  Call Extruder(6734.21438)
  MoveL 616 to (16.69, 20.93, 35) mm, rotated rx -180 ry 0 rz 180 deg; joints [-158.019, -62.995, -84.833, 25.494, 60.412, -13.249]
  Call Extruder(6743.57930)
  MoveL 617 to (11.61, 24.11, 35) mm, rotated rx -180 ry 0 rz 180 deg; joints [-157.299, -62.811, -85.449, 26.193, 60.967, -13.427]
  Call Extruder(6752.94410)
  MoveL 618 to (5.96, 26.09, 35) mm, rotated rx 180 ry 0 rz 180 deg; joints [-156.697, -62.583, -86.227, 26.726, 61.599, -13.468]
  Call Extruder(6762.30921)
  MoveL 619 to (0, 26.77, 35) mm, rotated rx -180 ry 0 rz 180 deg; joints [-156.245, -62.323, -87.131, 27.069, 62.279, -13.372]
  Call Extruder(6771.67431)
  MoveL 620 to (-5.96, 26.09, 35) mm, rotated rx 180 ry 0 rz 180 deg; joints [-155.969, -62.047, -88.117, 27.203, 62.974, -13.147]
  Call Extruder(6781.03910)
  MoveL 621 to (-11.61, 24.12, 35) mm, rotated rx 180 ry 0 rz 180 deg; joints [-155.891, -61.768, -89.137, 27.118, 63.651, -12.806]
  Call Extruder(6790.40402)
  MoveL 622 to (-16.69, 20.93, 35) mm, rotated rx 180 ry 0 rz -180 deg; joints [-156.025, -61.503, -90.14, 26.81, 64.279, -12.37]
  Call Extruder(6799.76923)
  MoveL 623 to (-20.93, 16.69, 35) mm, rotated rx 180 ry 0 rz 180 deg; joints [-156.374, -61.262, -91.076, 26.284, 64.828, -11.863]
  Call Extruder(6809.13414)
  MoveL 624 to (-24.11, 11.61, 35) mm, rotated rx -180 ry 0 rz 180 deg; joints [-156.928, -61.058, -91.897, 25.56, 65.271, -11.314]
  Call Extruder(6818.49894)
  MoveL 625 to (-26.09, 5.96, 35) mm, rotated rx -180 ry 0 rz 180 deg; joints [-157.665, -60.897, -92.558, 24.667, 65.583, -10.749]
  Call Extruder(6827.86405)
  MoveL 626 to (-26.77, 0, 35) mm, rotated rx 180 ry 0 rz 180 deg; joints [-158.546, -60.787, -93.024, 23.65, 65.748, -10.198]
  Call Extruder(6832.65278)
  MoveL 627 to (-26.42, -3.05, 35) mm, rotated rx -180 ry 0 rz 180 deg; joints [-159.044, -60.757, -93.152, 23.095, 65.75, -9.934]
  Set speed (130.0 mm/s)
  MoveL 628 to (-41.86, -6.29, 35) mm, rotated rx 180 ry 0 rz -180 deg; joints [-158.606, -60.2, -95.665, 23.234, 67.622, -9.283]
  Call Extruder(6837.65063)
  Set speed (60.0 mm/s)
  MoveL 629 to (-41.5, -9.47, 35) mm, rotated rx 180 ry 0 rz 180 deg; joints [-159.151, -60.173, -95.794, 22.635, 67.63, -9.018]
  Call Extruder(6852.54627)
  MoveL 630 to (-38.36, -18.47, 35) mm, rotated rx 180 ry 0 rz -180 deg; joints [-160.835, -60.169, -95.813, 20.831, 67.39, -8.322]
  Call Extruder(6867.44213)
  MoveL 631 to (-33.29, -26.54, 35) mm, rotated rx 180 ry 0 rz -180 deg; joints [-162.466, -60.245, -95.451, 19.121, 66.892, -7.748]
  Call Extruder(6882.33794)
  MoveL 632 to (-26.54, -33.28, 35) mm, rotated rx -180 ry 0 rz -180 deg; joints [-163.93, -60.4, -94.729, 17.616, 66.162, -7.313]
  Call Extruder(6897.23380)
  MoveL 633 to (-18.47, -38.36, 35) mm, rotated rx 180 ry 0 rz 180 deg; joints [-165.137, -60.632, -93.69, 16.408, 65.24, -7.031]
  Call Extruder(6912.12945)
  MoveL 634 to (-9.47, -41.5, 35) mm, rotated rx 180 ry 0 rz 180 deg; joints [-166.024, -60.937, -92.392, 15.563, 64.178, -6.917]
  Call Extruder(6927.02533)
  MoveL 635 to (0, -42.57, 35) mm, rotated rx 180 ry 0 rz 180 deg; joints [-166.562, -61.305, -90.908, 15.114, 63.036, -6.982]
  Call Extruder(6928.24069)
  MoveL 636 to (0.77, -42.49, 35) mm, rotated rx 180 ry 0 rz 180 deg; joints [-166.577, -61.338, -90.779, 15.11, 62.942, -7.002]
  Call Extruder(6941.92120)
  MoveL 637 to (9.47, -41.51, 35) mm, rotated rx 180 ry 0 rz 180 deg; joints [-166.745, -61.721, -89.315, 15.069, 61.877, -7.233]
  Call Extruder(6956.81686)
  MoveL 638 to (18.47, -38.36, 35) mm, rotated rx 180 ry 0 rz 180 deg; joints [-166.591, -62.165, -87.694, 15.412, 60.761, -7.669]
  Call Extruder(6971.71270)
  MoveL 639 to (26.54, -33.28, 35) mm, rotated rx 180 ry 0 rz 180 deg; joints [-166.133, -62.613, -86.123, 16.109, 59.745, -8.279]
  Call Extruder(6986.60852)
  MoveL 640 to (33.29, -26.54, 35) mm, rotated rx -180 ry 0 rz 180 deg; joints [-165.409, -63.041, -84.679, 17.113, 58.88, -9.041]
  Call Extruder(7001.50437)
  MoveL 641 to (38.36, -18.47, 35) mm, rotated rx 180 ry 0 rz 180 deg; joints [-164.468, -63.423, -83.43, 18.364, 58.208, -9.92]
  Call Extruder(7016.40003)
  MoveL 642 to (41.5, -9.47, 35) mm, rotated rx 180 ry 0 rz 180 deg; joints [-163.355, -63.734, -82.433, 19.795, 57.761, -10.868]
  Call Extruder(7031.29590)
  MoveL 643 to (42.57, 0, 35) mm, rotated rx 180 ry 0 rz 180 deg; joints [-162.12, -63.955, -81.735, 21.334, 57.558, -11.833]
  Call Extruder(7046.19177)
  MoveL 644 to (41.5, 9.47, 35) mm, rotated rx 180 ry 0 rz 180 deg; joints [-160.81, -64.073, -81.369, 22.909, 57.606, -12.757]
  Call Extruder(7061.08744)
  MoveL 645 to (38.36, 18.47, 35) mm, rotated rx 180 ry 0 rz 180 deg; joints [-159.475, -64.078, -81.351, 24.45, 57.9, -13.583]
  Call Extruder(7075.98328)
  MoveL 646 to (33.29, 26.54, 35) mm, rotated rx 180 ry 0 rz 180 deg; joints [-158.16, -63.972, -81.683, 25.892, 58.42, -14.262]
  Call Extruder(7090.87910)
  MoveL 647 to (26.54, 33.28, 35) mm, rotated rx -180 ry 0 rz 180 deg; joints [-156.916, -63.76, -82.349, 27.178, 59.139, -14.755]
  Call Extruder(7105.77495)
  MoveL 648 to (18.47, 38.36, 35) mm, rotated rx -180 ry 0 rz -180 deg; joints [-155.789, -63.457, -83.319, 28.259, 60.018, -15.035]
  Call Extruder(7120.67061)
  MoveL 649 to (9.47, 41.51, 35) mm, rotated rx -180 ry 0 rz 180 deg; joints [-154.828, -63.081, -84.546, 29.094, 61.015, -15.091]
  Call Extruder(7135.56648)
  MoveL 650 to (0, 42.57, 35) mm, rotated rx 180 ry 0 rz 180 deg; joints [-154.081, -62.657, -85.973, 29.648, 62.083, -14.922]
  Call Extruder(7150.46236)
  MoveL 651 to (-9.47, 41.51, 35) mm, rotated rx 180 ry 0 rz 180 deg; joints [-153.594, -62.209, -87.534, 29.892, 63.173, -14.543]
  Call Extruder(7165.35801)
  MoveL 652 to (-18.47, 38.36, 35) mm, rotated rx 180 ry 0 rz 180 deg; joints [-153.408, -61.764, -89.154, 29.804, 64.237, -13.98]
  Call Extruder(7180.25386)
  MoveL 653 to (-26.54, 33.28, 35) mm, rotated rx 180 ry 0 rz -180 deg; joints [-153.557, -61.344, -90.754, 29.369, 65.228, -13.268]
  Call Extruder(7195.14968)
  MoveL 654 to (-33.29, 26.54, 35) mm, rotated rx -180 ry 0 rz 180 deg; joints [-154.059, -60.971, -92.252, 28.585, 66.101, -12.448]
  Call Extruder(7210.04552)
  MoveL 655 to (-38.36, 18.47, 35) mm, rotated rx 180 ry 0 rz 180 deg; joints [-154.913, -60.659, -93.571, 27.468, 66.813, -11.568]
  Call Extruder(7224.94118)
  MoveL 656 to (-41.5, 9.47, 35) mm, rotated rx 180 ry 0 rz 180 deg; joints [-156.091, -60.419, -94.639, 26.056, 67.325, -10.674]
  Call Extruder(7239.83706)
  MoveL 657 to (-42.57, 0, 35) mm, rotated rx -180 ry 0 rz -180 deg; joints [-157.533, -60.257, -95.395, 24.414, 67.605, -9.812]
  Call Extruder(7247.39133)
  MoveL 658 to (-42.03, -4.8, 35) mm, rotated rx 180 ry 0 rz 180 deg; joints [-158.35, -60.213, -95.603, 23.515, 67.618, -9.407]
  Set speed (130.0 mm/s)
  MoveL 659 to (-54.1, -7.67, 35) mm, rotated rx -180 ry 0 rz -180 deg; joints [-158.024, -59.828, -97.542, 23.615, 69.095, -8.867]
  Call Extruder(7251.46397)
  Set speed (30.0 mm/s)
  MoveL 660 to (-53.59, -12.23, 35) mm, rotated rx 180 ry 0 rz -180 deg; joints [-158.835, -59.793, -97.729, 22.734, 69.112, -8.497]
  Call Extruder(7262.39410)
  MoveL 661 to (-49.52, -23.85, 35) mm, rotated rx 180 ry 0 rz 180 deg; joints [-161.095, -59.788, -97.754, 20.333, 68.814, -7.628]
  Call Extruder(7273.32438)
  MoveL 662 to (-42.98, -34.27, 35) mm, rotated rx 180 ry 0 rz 180 deg; joints [-163.275, -59.878, -97.277, 18.059, 68.172, -6.913]
  Call Extruder(7284.25450)
  MoveL 663 to (-34.27, -42.98, 35) mm, rotated rx -180 ry 0 rz 180 deg; joints [-165.21, -60.064, -96.329, 16.073, 67.22, -6.366]
  Call Extruder(7295.18479)
  MoveL 664 to (-23.85, -49.53, 35) mm, rotated rx 180 ry 0 rz -180 deg; joints [-166.774, -60.347, -94.97, 14.502, 66.014, -6.003]
  Call Extruder(7306.11492)
  MoveL 665 to (-12.23, -53.59, 35) mm, rotated rx 180 ry 0 rz 180 deg; joints [-167.889, -60.727, -93.28, 13.427, 64.627, -5.841]
  Call Extruder(7317.04514)
  MoveL 666 to (0, -54.97, 35) mm, rotated rx 180 ry 0 rz 180 deg; joints [-168.526, -61.192, -91.354, 12.884, 63.139, -5.9]
  Call Extruder(7318.96829)
  MoveL 667 to (2.15, -54.73, 35) mm, rotated rx 180 ry 0 rz -180 deg; joints [-168.557, -61.283, -90.994, 12.88, 62.874, -5.952]
  Call Extruder(7327.97536)
  MoveL 668 to (12.23, -53.59, 35) mm, rotated rx -180 ry 0 rz 180 deg; joints [-168.697, -61.726, -89.294, 12.87, 61.634, -6.196]
  Call Extruder(7338.90550)
  MoveL 669 to (23.85, -49.53, 35) mm, rotated rx 180 ry 0 rz 180 deg; joints [-168.436, -62.303, -87.203, 13.358, 60.189, -6.732]
  Call Extruder(7349.83578)
  MoveL 670 to (34.27, -42.98, 35) mm, rotated rx 180 ry 0 rz -180 deg; joints [-167.797, -62.89, -85.184, 14.295, 58.877, -7.503]
  Call Extruder(7360.76590)
  MoveL 671 to (42.98, -34.27, 35) mm, rotated rx 180 ry 0 rz 180 deg; joints [-166.837, -63.454, -83.329, 15.618, 57.763, -8.481]
  Call Extruder(7371.69618)
  MoveL 672 to (49.53, -23.85, 35) mm, rotated rx -180 ry 0 rz 180 deg; joints [-165.618, -63.958, -81.725, 17.247, 56.9, -9.622]
  Call Extruder(7382.62632)
  MoveL 673 to (53.59, -12.23, 35) mm, rotated rx 180 ry 0 rz -180 deg; joints [-164.2, -64.372, -80.446, 19.097, 56.33, -10.865]
  Call Extruder(7393.55654)
  MoveL 674 to (54.97, 0, 35) mm, rotated rx -180 ry 0 rz 180 deg; joints [-162.641, -64.667, -79.551, 21.074, 56.077, -12.137]
  Call Extruder(7404.48676)
  MoveL 675 to (53.59, 12.23, 35) mm, rotated rx -180 ry 0 rz 180 deg; joints [-160.996, -64.823, -79.081, 23.085, 56.149, -13.356]
  Call Extruder(7415.41691)
  MoveL 676 to (49.52, 23.85, 35) mm, rotated rx 180 ry 0 rz -180 deg; joints [-159.322, -64.831, -79.058, 25.041, 56.538, -14.445]
  Call Extruder(7426.34718)
  MoveL 677 to (42.98, 34.27, 35) mm, rotated rx -180 ry 0 rz 180 deg; joints [-157.673, -64.689, -79.485, 26.863, 57.217, -15.337]
  Call Extruder(7437.27731)
  MoveL 678 to (34.27, 42.98, 35) mm, rotated rx 180 ry 0 rz 180 deg; joints [-156.102, -64.407, -80.339, 28.484, 58.149, -15.979]
  Call Extruder(7448.20758)
  MoveL 679 to (23.85, 49.52, 35) mm, rotated rx -180 ry 0 rz 180 deg; joints [-154.667, -64.004, -81.583, 29.848, 59.282, -16.337]
  Call Extruder(7459.13773)
  MoveL 680 to (12.23, 53.59, 35) mm, rotated rx -180 ry 0 rz 180 deg; joints [-153.426, -63.507, -83.157, 30.909, 60.562, -16.397]
  Call Extruder(7470.06795)
  MoveL 681 to (0, 54.97, 35) mm, rotated rx 180 ry 0 rz 180 deg; joints [-152.438, -62.948, -84.991, 31.628, 61.928, -16.163]
  Call Extruder(7480.99817)
  MoveL 682 to (-12.23, 53.59, 35) mm, rotated rx -180 ry 0 rz 180 deg; joints [-151.764, -62.361, -86.998, 31.97, 63.32, -15.655]
  Call Extruder(7491.92830)
  MoveL 683 to (-23.85, 49.52, 35) mm, rotated rx 180 ry 0 rz 180 deg; joints [-151.463, -61.782, -89.086, 31.904, 64.68, -14.909]
  Call Extruder(7502.85859)
  MoveL 684 to (-34.27, 42.98, 35) mm, rotated rx -180 ry 0 rz 180 deg; joints [-151.589, -61.243, -91.154, 31.401, 65.949, -13.97]
  Call Extruder(7513.78871)
  MoveL 685 to (-42.98, 34.27, 35) mm, rotated rx 180 ry 0 rz -180 deg; joints [-152.179, -60.769, -93.098, 30.446, 67.074, -12.897]
  Call Extruder(7524.71899)
  MoveL 686 to (-49.52, 23.85, 35) mm, rotated rx 180 ry 0 rz 180 deg; joints [-153.248, -60.381, -94.816, 29.044, 68, -11.751]
  Call Extruder(7535.64913)
  MoveL 687 to (-53.59, 12.23, 35) mm, rotated rx 180 ry 0 rz 180 deg; joints [-154.769, -60.087, -96.212, 27.231, 68.678, -10.599]
  Call Extruder(7546.57935)
  MoveL 688 to (-54.97, 0, 35) mm, rotated rx -180 ry 0 rz -180 deg; joints [-156.673, -59.892, -97.203, 25.087, 69.06, -9.498]
  Call Extruder(7552.10496)
  MoveL 689 to (-54.27, -6.18, 35) mm, rotated rx -180 ry 0 rz 180 deg; joints [-157.76, -59.84, -97.478, 23.902, 69.088, -8.989]
  Set speed (130.0 mm/s)
  MoveL 690 to (-49.9, -9.51, 35) mm, rotated rx -180 ry 0 rz -180 deg; joints [-158.616, -59.924, -97.035, 23.05, 68.627, -8.815]
  MoveL 691 to (2.97, -12.99, 35) mm, rotated rx 180 ry 0 rz -180 deg; joints [-162.152, -61.783, -89.081, 20.235, 62.39, -9.695]
  Call Extruder(7556.76854)
  Set speed (80.0 mm/s)
  MoveL 692 to (5.78, -12.01, 35) mm, rotated rx -180 ry 0 rz 180 deg; joints [-162.141, -61.921, -88.573, 20.316, 62.045, -9.846]
  Call Extruder(7561.43216)
  MoveL 693 to (8.31, -10.42, 35) mm, rotated rx -180 ry 0 rz -180 deg; joints [-162.027, -62.058, -88.077, 20.51, 61.728, -10.048]
  Call Extruder(7566.09635)
  MoveL 694 to (10.42, -8.31, 35) mm, rotated rx 180 ry 0 rz 180 deg; joints [-161.819, -62.185, -87.619, 20.805, 61.455, -10.291]
  Call Extruder(7570.75998)
  MoveL 695 to (12.01, -5.78, 35) mm, rotated rx 180 ry 0 rz 180 deg; joints [-161.529, -62.298, -87.221, 21.187, 61.241, -10.564]
  Call Extruder(7575.42355)
  MoveL 696 to (12.99, -2.97, 35) mm, rotated rx 180 ry 0 rz -180 deg; joints [-161.171, -62.388, -86.903, 21.634, 61.096, -10.852]
  Call Extruder(7580.08750)
  MoveL 697 to (13.33, 0, 35) mm, rotated rx 180 ry 0 rz 180 deg; joints [-160.763, -62.452, -86.68, 22.124, 61.026, -11.141]
  Call Extruder(7584.75146)
  MoveL 698 to (13, 2.97, 35) mm, rotated rx 180 ry 0 rz 180 deg; joints [-160.324, -62.486, -86.563, 22.634, 61.035, -11.416]
  Call Extruder(7589.41503)
  MoveL 699 to (12.01, 5.78, 35) mm, rotated rx 180 ry 0 rz -180 deg; joints [-159.874, -62.488, -86.557, 23.139, 61.121, -11.661]
  Call Extruder(7594.07865)
  MoveL 700 to (10.42, 8.31, 35) mm, rotated rx -180 ry 0 rz 180 deg; joints [-159.432, -62.457, -86.663, 23.615, 61.28, -11.864]
  Call Extruder(7598.74284)
  MoveL 701 to (8.31, 10.42, 35) mm, rotated rx 180 ry 0 rz 180 deg; joints [-159.021, -62.396, -86.876, 24.041, 61.505, -12.014]
  Call Extruder(7603.40647)
  MoveL 702 to (5.78, 12.01, 35) mm, rotated rx 180 ry 0 rz 180 deg; joints [-158.657, -62.308, -87.186, 24.396, 61.782, -12.103]
  Call Extruder(7608.07004)
  MoveL 703 to (2.97, 12.99, 35) mm, rotated rx -180 ry 0 rz 180 deg; joints [-158.359, -62.197, -87.577, 24.663, 62.1, -12.126]
  Call Extruder(7612.73400)
  MoveL 704 to (0, 13.33, 35) mm, rotated rx 180 ry 0 rz -180 deg; joints [-158.143, -62.071, -88.03, 24.831, 62.442, -12.083]
  Call Extruder(7617.39795)
  MoveL 705 to (-2.97, 12.99, 35) mm, rotated rx -180 ry 0 rz 180 deg; joints [-158.019, -61.935, -88.523, 24.889, 62.792, -11.977]
  Call Extruder(7622.06151)
  MoveL 706 to (-5.78, 12.01, 35) mm, rotated rx 180 ry 0 rz 180 deg; joints [-157.997, -61.797, -89.031, 24.834, 63.132, -11.813]
  Call Extruder(7626.72515)
  MoveL 707 to (-8.31, 10.42, 35) mm, rotated rx -180 ry 0 rz 180 deg; joints [-158.08, -61.663, -89.53, 24.666, 63.447, -11.601]
  Call Extruder(7631.38934)
  MoveL 708 to (-10.42, 8.31, 35) mm, rotated rx 180 ry 0 rz 180 deg; joints [-158.266, -61.541, -89.993, 24.392, 63.72, -11.352]
  Call Extruder(7636.05296)
  MoveL 709 to (-12.01, 5.78, 35) mm, rotated rx 180 ry 0 rz 180 deg; joints [-158.549, -61.436, -90.398, 24.023, 63.938, -11.079]
  Call Extruder(7640.71653)
  MoveL 710 to (-13, 2.97, 35) mm, rotated rx -180 ry 0 rz -180 deg; joints [-158.913, -61.352, -90.723, 23.577, 64.09, -10.796]
  Call Extruder(7645.38049)
  MoveL 711 to (-13.33, 0, 35) mm, rotated rx -180 ry 0 rz 180 deg; joints [-159.341, -61.294, -90.952, 23.077, 64.168, -10.517]
  Call Extruder(7650.04444)
  MoveL 712 to (-13, -2.97, 35) mm, rotated rx -180 ry 0 rz 180 deg; joints [-159.811, -61.263, -91.072, 22.547, 64.166, -10.255]
  Call Extruder(7654.70800)
  MoveL 713 to (-12.01, -5.78, 35) mm, rotated rx -180 ry 0 rz 180 deg; joints [-160.294, -61.262, -91.078, 22.017, 64.085, -10.022]
  Call Extruder(7659.37164)
  MoveL 714 to (-10.42, -8.31, 35) mm, rotated rx 180 ry 0 rz 180 deg; joints [-160.766, -61.289, -90.969, 21.515, 63.928, -9.829]
  Call Extruder(7664.03583)
  MoveL 715 to (-8.31, -10.42, 35) mm, rotated rx 180 ry 0 rz 180 deg; joints [-161.2, -61.345, -90.75, 21.068, 63.702, -9.685]
  Call Extruder(7668.69946)
  MoveL 716 to (-5.78, -12.01, 35) mm, rotated rx 180 ry 0 rz 180 deg; joints [-161.572, -61.426, -90.434, 20.7, 63.421, -9.597]
  Call Extruder(7673.36302)
  MoveL 717 to (-2.97, -13, 35) mm, rotated rx 180 ry 0 rz 180 deg; joints [-161.863, -61.53, -90.036, 20.431, 63.097, -9.568]
  Call Extruder(7678.02699)
  MoveL 718 to (0, -13.33, 35) mm, rotated rx -180 ry 0 rz -180 deg; joints [-162.059, -61.651, -89.577, 20.274, 62.747, -9.601]
  Call Extruder(7682.69093)
  MoveL 719 to (2.97, -12.99, 35) mm, rotated rx 180 ry 0 rz -180 deg; joints [-162.152, -61.783, -89.081, 20.235, 62.39, -9.695]
  Set speed (130.0 mm/s)
  MoveL 720 to (2.97, -12.99, 40) mm, rotated rx 180 ry 0 rz -180 deg; joints [-162.152, -61.016, -89.511, 20.297, 62.074, -9.827]
  MoveL 721 to (-26.25, -4.54, 40) mm, rotated rx 180 ry 0 rz -180 deg; joints [-159.288, -59.949, -93.651, 22.886, 65.424, -9.957]
  Call Extruder(7684.92356)
  Set speed (60.0 mm/s)
  MoveL 722 to (-26.09, -5.96, 40) mm, rotated rx 180 ry 0 rz 180 deg; joints [-159.522, -59.936, -93.708, 22.625, 65.424, -9.834]
  Call Extruder(7694.28835)
  MoveL 723 to (-24.11, -11.61, 40) mm, rotated rx 180 ry 0 rz 180 deg; joints [-160.532, -59.933, -93.72, 21.528, 65.264, -9.373]
  Call Extruder(7703.65327)
  MoveL 724 to (-20.93, -16.69, 40) mm, rotated rx 180 ry 0 rz -180 deg; joints [-161.513, -59.986, -93.496, 20.488, 64.949, -8.991]
  Call Extruder(7713.01847)
  MoveL 725 to (-16.69, -20.93, 40) mm, rotated rx 180 ry 0 rz 180 deg; joints [-162.406, -60.095, -93.05, 19.567, 64.494, -8.702]
  Call Extruder(7722.38339)
  MoveL 726 to (-11.61, -24.12, 40) mm, rotated rx 180 ry 0 rz 180 deg; joints [-163.159, -60.254, -92.405, 18.817, 63.923, -8.519]
  Call Extruder(7731.74818)
  MoveL 727 to (-5.96, -26.09, 40) mm, rotated rx 180 ry 0 rz 180 deg; joints [-163.733, -60.46, -91.597, 18.278, 63.267, -8.451]
  Call Extruder(7741.11329)
  MoveL 728 to (0, -26.77, 40) mm, rotated rx 180 ry 0 rz 180 deg; joints [-164.103, -60.703, -90.669, 17.977, 62.561, -8.504]
  Call Extruder(7745.37891)
  MoveL 729 to (2.71, -26.46, 40) mm, rotated rx -180 ry 0 rz -180 deg; joints [-164.174, -60.824, -90.215, 17.951, 62.234, -8.583]
  Call Extruder(7750.47839)
  MoveL 730 to (5.96, -26.09, 40) mm, rotated rx 180 ry 0 rz -180 deg; joints [-164.258, -60.973, -89.668, 17.922, 61.843, -8.677]
  Call Extruder(7759.84319)
  MoveL 731 to (11.61, -24.11, 40) mm, rotated rx 180 ry 0 rz 180 deg; joints [-164.201, -61.256, -88.646, 18.111, 61.149, -8.968]
  Call Extruder(7769.20811)
  MoveL 732 to (16.69, -20.93, 40) mm, rotated rx 180 ry 0 rz 180 deg; joints [-163.944, -61.539, -87.653, 18.526, 60.516, -9.365]
  Call Extruder(7778.57331)
  MoveL 733 to (20.93, -16.69, 40) mm, rotated rx -180 ry 0 rz 180 deg; joints [-163.508, -61.806, -86.738, 19.14, 59.975, -9.852]
  Call Extruder(7787.93823)
  MoveL 734 to (24.12, -11.61, 40) mm, rotated rx -180 ry 0 rz 180 deg; joints [-162.92, -62.042, -85.944, 19.919, 59.553, -10.405]
  Call Extruder(7797.30303)
  MoveL 735 to (26.09, -5.96, 40) mm, rotated rx -180 ry 0 rz -180 deg; joints [-162.209, -62.234, -85.311, 20.821, 59.271, -10.996]
  Call Extruder(7806.66813)
  MoveL 736 to (26.77, 0, 40) mm, rotated rx -180 ry 0 rz -180 deg; joints [-161.41, -62.37, -84.867, 21.8, 59.14, -11.594]
  Call Extruder(7816.03323)
  MoveL 737 to (26.09, 5.96, 40) mm, rotated rx -180 ry 0 rz 180 deg; joints [-160.556, -62.441, -84.634, 22.81, 59.167, -12.164]
  Call Extruder(7825.39804)
  MoveL 738 to (24.12, 11.61, 40) mm, rotated rx 180 ry 0 rz 180 deg; joints [-159.683, -62.445, -84.623, 23.804, 59.348, -12.675]
  Call Extruder(7834.76295)
  MoveL 739 to (20.93, 16.69, 40) mm, rotated rx -180 ry 0 rz 180 deg; joints [-158.826, -62.38, -84.834, 24.738, 59.672, -13.097]
  Call Extruder(7844.12816)
  MoveL 740 to (16.69, 20.93, 40) mm, rotated rx -180 ry 0 rz 180 deg; joints [-158.019, -62.25, -85.258, 25.573, 60.123, -13.408]
  Call Extruder(7853.49307)
  MoveL 741 to (11.61, 24.11, 40) mm, rotated rx -180 ry 0 rz 180 deg; joints [-157.299, -62.063, -85.874, 26.272, 60.678, -13.59]
  Call Extruder(7862.85787)
  MoveL 742 to (5.96, 26.09, 40) mm, rotated rx 180 ry 0 rz 180 deg; joints [-156.697, -61.831, -86.653, 26.805, 61.308, -13.635]
  Call Extruder(7872.22298)
  MoveL 743 to (0, 26.77, 40) mm, rotated rx -180 ry 0 rz 180 deg; joints [-156.245, -61.566, -87.558, 27.148, 61.985, -13.542]
  Call Extruder(7881.58808)
  MoveL 744 to (-5.96, 26.09, 40) mm, rotated rx 180 ry 0 rz 180 deg; joints [-155.969, -61.284, -88.546, 27.282, 62.677, -13.318]
  Call Extruder(7890.95287)
  MoveL 745 to (-11.61, 24.12, 40) mm, rotated rx -180 ry 0 rz 180 deg; joints [-155.891, -61, -89.567, 27.195, 63.35, -12.978]
  Call Extruder(7900.31779)
  MoveL 746 to (-16.69, 20.93, 40) mm, rotated rx 180 ry 0 rz -180 deg; joints [-156.025, -60.729, -90.572, 26.885, 63.974, -12.542]
  Call Extruder(7909.68300)
  MoveL 747 to (-20.93, 16.69, 40) mm, rotated rx 180 ry 0 rz -180 deg; joints [-156.374, -60.483, -91.51, 26.357, 64.518, -12.033]
  Call Extruder(7919.04791)
  MoveL 748 to (-24.11, 11.61, 40) mm, rotated rx 180 ry 0 rz 180 deg; joints [-156.928, -60.273, -92.332, 25.63, 64.956, -11.48]
  Call Extruder(7928.41271)
  MoveL 749 to (-26.09, 5.96, 40) mm, rotated rx 180 ry 0 rz 180 deg; joints [-157.665, -60.108, -92.994, 24.735, 65.263, -10.911]
  Call Extruder(7937.77782)
  MoveL 750 to (-26.77, 0, 40) mm, rotated rx 180 ry 0 rz -180 deg; joints [-158.546, -59.995, -93.462, 23.715, 65.423, -10.354]
  Call Extruder(7942.56655)
  MoveL 751 to (-26.42, -3.05, 40) mm, rotated rx 180 ry 0 rz 180 deg; joints [-159.044, -59.964, -93.59, 23.159, 65.424, -10.087]
  Set speed (130.0 mm/s)
  MoveL 752 to (-41.86, -6.3, 40) mm, rotated rx 180 ry 0 rz 180 deg; joints [-158.606, -59.39, -96.109, 23.294, 67.286, -9.439]
  Call Extruder(7947.56440)
  Set speed (60.0 mm/s)
  MoveL 753 to (-41.5, -9.47, 40) mm, rotated rx -180 ry 0 rz -180 deg; joints [-159.151, -59.362, -96.238, 22.694, 67.291, -9.171]
  Call Extruder(7962.46005)
  MoveL 754 to (-38.36, -18.47, 40) mm, rotated rx 180 ry 0 rz 180 deg; joints [-160.835, -59.358, -96.257, 20.886, 67.047, -8.464]
  Call Extruder(7977.35590)
  MoveL 755 to (-33.29, -26.54, 40) mm, rotated rx 180 ry 0 rz 180 deg; joints [-162.466, -59.436, -95.894, 19.172, 66.547, -7.878]
  Call Extruder(7992.25172)
  MoveL 756 to (-26.54, -33.28, 40) mm, rotated rx 180 ry 0 rz -180 deg; joints [-163.93, -59.596, -95.17, 17.665, 65.817, -7.433]
  Call Extruder(8007.14757)
  MoveL 757 to (-18.47, -38.36, 40) mm, rotated rx 180 ry 0 rz 180 deg; joints [-165.137, -59.836, -94.128, 16.455, 64.897, -7.142]
  Call Extruder(8022.04322)
  MoveL 758 to (-9.47, -41.51, 40) mm, rotated rx -180 ry 0 rz 180 deg; joints [-166.024, -60.149, -92.828, 15.609, 63.839, -7.022]
  Call Extruder(8036.93910)
  MoveL 759 to (0, -42.57, 40) mm, rotated rx 180 ry 0 rz -180 deg; joints [-166.562, -60.526, -91.341, 15.16, 62.703, -7.083]
  Call Extruder(8043.97027)
  MoveL 760 to (4.47, -42.07, 40) mm, rotated rx 180 ry 0 rz 180 deg; joints [-166.65, -60.724, -90.591, 15.137, 62.158, -7.201]
  Call Extruder(8051.83497)
  MoveL 761 to (9.47, -41.51, 40) mm, rotated rx -180 ry 0 rz 180 deg; joints [-166.745, -60.951, -89.745, 15.116, 61.55, -7.333]
  Call Extruder(8066.73063)
  MoveL 762 to (18.47, -38.36, 40) mm, rotated rx -180 ry 0 rz 180 deg; joints [-166.591, -61.405, -88.122, 15.462, 60.441, -7.77]
  Call Extruder(8081.62648)
  MoveL 763 to (26.54, -33.29, 40) mm, rotated rx 180 ry 0 rz 180 deg; joints [-166.133, -61.862, -86.549, 16.162, 59.433, -8.384]
  Call Extruder(8096.52230)
  MoveL 764 to (33.29, -26.54, 40) mm, rotated rx 180 ry 0 rz 180 deg; joints [-165.409, -62.297, -85.104, 17.17, 58.575, -9.152]
  Call Extruder(8111.41815)
  MoveL 765 to (38.36, -18.47, 40) mm, rotated rx -180 ry 0 rz 180 deg; joints [-164.468, -62.684, -83.853, 18.426, 57.91, -10.037]
  Call Extruder(8126.31380)
  MoveL 766 to (41.51, -9.47, 40) mm, rotated rx 180 ry 0 rz 180 deg; joints [-163.355, -63, -82.855, 19.862, 57.469, -10.993]
  Call Extruder(8141.20967)
  MoveL 767 to (42.57, 0, 40) mm, rotated rx 180 ry 0 rz 180 deg; joints [-162.12, -63.225, -82.157, 21.406, 57.271, -11.967]
  Call Extruder(8156.10555)
  MoveL 768 to (41.5, 9.47, 40) mm, rotated rx -180 ry 0 rz 180 deg; joints [-160.81, -63.344, -81.791, 22.985, 57.324, -12.899]
  Call Extruder(8171.00121)
  MoveL 769 to (38.36, 18.47, 40) mm, rotated rx 180 ry 0 rz 180 deg; joints [-159.475, -63.35, -81.773, 24.53, 57.621, -13.733]
  Call Extruder(8185.89705)
  MoveL 770 to (33.29, 26.54, 40) mm, rotated rx 180 ry 0 rz 180 deg; joints [-158.16, -63.242, -82.105, 25.975, 58.143, -14.421]
  Call Extruder(8200.79288)
  MoveL 771 to (26.54, 33.28, 40) mm, rotated rx -180 ry 0 rz 180 deg; joints [-156.916, -63.027, -82.772, 27.263, 58.863, -14.921]
  Call Extruder(8215.68872)
  MoveL 772 to (18.47, 38.36, 40) mm, rotated rx -180 ry 0 rz -180 deg; joints [-155.789, -62.719, -83.742, 28.345, 59.741, -15.208]
  Call Extruder(8230.58439)
  MoveL 773 to (9.47, 41.51, 40) mm, rotated rx -180 ry 0 rz -180 deg; joints [-154.828, -62.338, -84.97, 29.18, 60.736, -15.268]
  Call Extruder(8245.48026)
  MoveL 774 to (0, 42.57, 40) mm, rotated rx 180 ry 0 rz 180 deg; joints [-154.081, -61.906, -86.399, 29.734, 61.8, -15.104]
  Call Extruder(8260.37613)
  MoveL 775 to (-9.47, 41.51, 40) mm, rotated rx -180 ry 0 rz 180 deg; joints [-153.594, -61.45, -87.962, 29.976, 62.886, -14.729]
  Call Extruder(8275.27178)
  MoveL 776 to (-18.47, 38.36, 40) mm, rotated rx -180 ry 0 rz 180 deg; joints [-153.408, -60.996, -89.584, 29.886, 63.944, -14.167]
  Call Extruder(8290.16764)
  MoveL 777 to (-26.54, 33.29, 40) mm, rotated rx 180 ry 0 rz 180 deg; joints [-153.557, -60.567, -91.186, 29.448, 64.928, -13.455]
  Call Extruder(8305.06345)
  MoveL 778 to (-33.28, 26.54, 40) mm, rotated rx 180 ry 0 rz 180 deg; joints [-154.059, -60.184, -92.688, 28.66, 65.793, -12.633]
  Call Extruder(8319.95930)
  MoveL 779 to (-38.36, 18.47, 40) mm, rotated rx 180 ry 0 rz 180 deg; joints [-154.913, -59.864, -94.01, 27.539, 66.496, -11.747]
  Call Extruder(8334.85496)
  MoveL 780 to (-41.51, 9.47, 40) mm, rotated rx -180 ry 0 rz -180 deg; joints [-156.091, -59.617, -95.08, 26.122, 67, -10.847]
  Call Extruder(8349.75083)
  MoveL 781 to (-42.57, 0, 40) mm, rotated rx 180 ry 0 rz -180 deg; joints [-157.533, -59.449, -95.838, 24.477, 67.273, -9.975]
  Call Extruder(8357.30511)
  MoveL 782 to (-42.03, -4.8, 40) mm, rotated rx 180 ry 0 rz -180 deg; joints [-158.35, -59.403, -96.046, 23.575, 67.283, -9.566]
  Set speed (130.0 mm/s)
  MoveL 783 to (-54.1, -7.67, 40) mm, rotated rx 180 ry 0 rz -180 deg; joints [-158.024, -59.005, -97.99, 23.673, 68.751, -9.028]
  Call Extruder(8361.37774)
  Set speed (30.0 mm/s)
  MoveL 784 to (-53.59, -12.23, 40) mm, rotated rx 180 ry 0 rz 180 deg; joints [-158.835, -58.968, -98.178, 22.79, 68.766, -8.652]
  Call Extruder(8372.30787)
  MoveL 785 to (-49.52, -23.85, 40) mm, rotated rx -180 ry 0 rz -180 deg; joints [-161.095, -58.964, -98.203, 20.385, 68.462, -7.768]
  Call Extruder(8383.23816)
  MoveL 786 to (-42.98, -34.27, 40) mm, rotated rx 180 ry 0 rz 180 deg; joints [-163.275, -59.057, -97.725, 18.106, 67.818, -7.038]
  Call Extruder(8394.16828)
  MoveL 787 to (-34.27, -42.98, 40) mm, rotated rx 180 ry 0 rz 180 deg; joints [-165.21, -59.249, -96.775, 16.117, 66.865, -6.477]
  Call Extruder(8405.09856)
  MoveL 788 to (-23.85, -49.53, 40) mm, rotated rx -180 ry 0 rz 180 deg; joints [-166.774, -59.542, -95.412, 14.543, 65.662, -6.102]
  Call Extruder(8416.02869)
  MoveL 789 to (-12.23, -53.59, 40) mm, rotated rx 180 ry 0 rz 180 deg; joints [-167.889, -59.933, -93.718, 13.467, 64.281, -5.933]
  Call Extruder(8426.95892)
  MoveL 790 to (0, -54.97, 40) mm, rotated rx 180 ry 0 rz 180 deg; joints [-168.526, -60.411, -91.788, 12.923, 62.801, -5.987]
  Call Extruder(8432.18725)
  MoveL 791 to (5.85, -54.31, 40) mm, rotated rx -180 ry 0 rz 180 deg; joints [-168.609, -60.667, -90.806, 12.915, 62.084, -6.128]
  Call Extruder(8437.88914)
  MoveL 792 to (12.23, -53.59, 40) mm, rotated rx 180 ry 0 rz 180 deg; joints [-168.697, -60.957, -89.724, 12.911, 61.304, -6.282]
  Call Extruder(8448.81928)
  MoveL 793 to (23.85, -49.53, 40) mm, rotated rx 180 ry 0 rz 180 deg; joints [-168.436, -61.545, -87.631, 13.402, 59.868, -6.821]
  Call Extruder(8459.74956)
  MoveL 794 to (34.27, -42.98, 40) mm, rotated rx -180 ry 0 rz 180 deg; joints [-167.797, -62.143, -85.609, 14.344, 58.565, -7.596]
  Call Extruder(8470.67968)
  MoveL 795 to (42.98, -34.27, 40) mm, rotated rx 180 ry 0 rz -180 deg; joints [-166.837, -62.716, -83.752, 15.671, 57.46, -8.581]
  Call Extruder(8481.60996)
  MoveL 796 to (49.53, -23.85, 40) mm, rotated rx 180 ry 0 rz 180 deg; joints [-165.618, -63.228, -82.147, 17.307, 56.606, -9.732]
  Call Extruder(8492.54010)
  MoveL 797 to (53.59, -12.23, 40) mm, rotated rx 180 ry 0 rz -180 deg; joints [-164.2, -63.647, -80.868, 19.163, 56.044, -10.985]
  Call Extruder(8503.47032)
  MoveL 798 to (54.97, 0, 40) mm, rotated rx 180 ry 0 rz 180 deg; joints [-162.641, -63.946, -79.972, 21.147, 55.798, -12.267]
  Call Extruder(8514.40054)
  MoveL 799 to (53.59, 12.23, 40) mm, rotated rx 180 ry 0 rz 180 deg; joints [-160.996, -64.104, -79.502, 23.164, 55.876, -13.497]
  Call Extruder(8525.33068)
  MoveL 800 to (49.52, 23.85, 40) mm, rotated rx 180 ry 0 rz -180 deg; joints [-159.322, -64.112, -79.48, 25.125, 56.268, -14.597]
  Call Extruder(8536.26096)
  MoveL 801 to (42.98, 34.27, 40) mm, rotated rx -180 ry 0 rz 180 deg; joints [-157.673, -63.968, -79.906, 26.951, 56.951, -15.498]
  Call Extruder(8547.19108)
  MoveL 802 to (34.27, 42.98, 40) mm, rotated rx 180 ry 0 rz 180 deg; joints [-156.102, -63.683, -80.761, 28.575, 57.883, -16.149]
  Call Extruder(8558.12136)
  MoveL 803 to (23.85, 49.52, 40) mm, rotated rx 180 ry 0 rz 180 deg; joints [-154.667, -63.274, -82.005, 29.94, 59.015, -16.515]
  Call Extruder(8569.05150)
  MoveL 804 to (12.23, 53.59, 40) mm, rotated rx 180 ry 0 rz 180 deg; joints [-153.426, -62.77, -83.58, 31.001, 60.293, -16.582]
  Call Extruder(8579.98172)
  MoveL 805 to (0, 54.97, 40) mm, rotated rx -180 ry 0 rz 180 deg; joints [-152.438, -62.202, -85.416, 31.719, 61.655, -16.354]
  Call Extruder(8590.91195)
  MoveL 806 to (-12.23, 53.59, 40) mm, rotated rx -180 ry 0 rz 180 deg; joints [-151.764, -61.605, -87.425, 32.059, 63.041, -15.851]
  Call Extruder(8601.84208)
  MoveL 807 to (-23.85, 49.52, 40) mm, rotated rx 180 ry 0 rz 180 deg; joints [-151.463, -61.014, -89.516, 31.989, 64.393, -15.107]
  Call Extruder(8612.77236)
  MoveL 808 to (-34.27, 42.98, 40) mm, rotated rx 180 ry 0 rz 180 deg; joints [-151.589, -60.463, -91.587, 31.482, 65.654, -14.168]
  Call Extruder(8623.70248)
  MoveL 809 to (-42.98, 34.27, 40) mm, rotated rx -180 ry 0 rz -180 deg; joints [-152.179, -59.977, -93.535, 30.523, 66.768, -13.092]
  Call Extruder(8634.63276)
  MoveL 810 to (-49.53, 23.85, 40) mm, rotated rx 180 ry 0 rz 180 deg; joints [-153.248, -59.577, -95.257, 29.116, 67.683, -11.942]
  Call Extruder(8645.56290)
  MoveL 811 to (-53.59, 12.23, 40) mm, rotated rx 180 ry 0 rz -180 deg; joints [-154.769, -59.274, -96.657, 27.298, 68.35, -10.78]
  Call Extruder(8656.49312)
  MoveL 812 to (-54.97, 0, 40) mm, rotated rx 180 ry 0 rz -180 deg; joints [-156.673, -59.071, -97.651, 25.148, 68.723, -9.668]
  Call Extruder(8662.01874)
  MoveL 813 to (-54.27, -6.18, 40) mm, rotated rx 180 ry 0 rz 180 deg; joints [-157.76, -59.017, -97.927, 23.961, 68.746, -9.152]
  Set speed (130.0 mm/s)
  MoveL 814 to (-49.9, -9.51, 40) mm, rotated rx 180 ry 0 rz 180 deg; joints [-158.616, -59.105, -97.482, 23.108, 68.284, -8.972]
  MoveL 815 to (1.22, -13.19, 40) mm, rotated rx -180 ry 0 rz 180 deg; joints [-162.097, -60.935, -89.805, 20.319, 62.283, -9.772]
  Call Extruder(8664.76778)
  Set speed (80.0 mm/s)
  MoveL 816 to (2.97, -12.99, 40) mm, rotated rx 180 ry 0 rz -180 deg; joints [-162.152, -61.016, -89.511, 20.297, 62.074, -9.827]
  Call Extruder(8669.43135)
  MoveL 817 to (5.78, -12.01, 40) mm, rotated rx 180 ry 0 rz 180 deg; joints [-162.141, -61.156, -89.002, 20.378, 61.73, -9.978]
  Call Extruder(8674.09498)
  MoveL 818 to (8.31, -10.42, 40) mm, rotated rx 180 ry 0 rz -180 deg; joints [-162.027, -61.296, -88.506, 20.573, 61.415, -10.181]
  Call Extruder(8678.75917)
  MoveL 819 to (10.42, -8.31, 40) mm, rotated rx -180 ry 0 rz 180 deg; joints [-161.819, -61.426, -88.047, 20.87, 61.146, -10.425]
  Call Extruder(8683.42279)
  MoveL 820 to (12.01, -5.78, 40) mm, rotated rx 180 ry 0 rz 180 deg; joints [-161.529, -61.54, -87.649, 21.253, 60.934, -10.7]
  Call Extruder(8688.08636)
  MoveL 821 to (12.99, -2.97, 40) mm, rotated rx -180 ry 0 rz -180 deg; joints [-161.171, -61.633, -87.33, 21.701, 60.79, -10.991]
  Call Extruder(8692.75032)
  MoveL 822 to (13.33, 0, 40) mm, rotated rx 180 ry 0 rz 180 deg; joints [-160.763, -61.698, -87.107, 22.193, 60.722, -11.283]
  Call Extruder(8697.41427)
  MoveL 823 to (13, 2.97, 40) mm, rotated rx 180 ry 0 rz 180 deg; joints [-160.324, -61.732, -86.989, 22.704, 60.733, -11.56]
  Call Extruder(8702.07785)
  MoveL 824 to (12.01, 5.78, 40) mm, rotated rx 180 ry 0 rz -180 deg; joints [-159.874, -61.734, -86.984, 23.21, 60.82, -11.809]
  Call Extruder(8706.74147)
  MoveL 825 to (10.42, 8.31, 40) mm, rotated rx 180 ry 0 rz 180 deg; joints [-159.432, -61.703, -87.09, 23.688, 60.98, -12.015]
  Call Extruder(8711.40566)
  MoveL 826 to (8.31, 10.42, 40) mm, rotated rx 180 ry 0 rz 180 deg; joints [-159.021, -61.64, -87.303, 24.114, 61.205, -12.167]
  Call Extruder(8716.06929)
  MoveL 827 to (5.78, 12.01, 40) mm, rotated rx 180 ry 0 rz 180 deg; joints [-158.657, -61.551, -87.613, 24.469, 61.482, -12.258]
  Call Extruder(8720.73286)
  MoveL 828 to (2.97, 13, 40) mm, rotated rx 180 ry 0 rz 180 deg; joints [-158.359, -61.438, -88.004, 24.737, 61.799, -12.283]
  Call Extruder(8725.39681)
  MoveL 829 to (0, 13.33, 40) mm, rotated rx 180 ry 0 rz 180 deg; joints [-158.143, -61.309, -88.458, 24.905, 62.14, -12.242]
  Call Extruder(8730.06077)
  MoveL 830 to (-2.97, 12.99, 40) mm, rotated rx -180 ry 0 rz 180 deg; joints [-158.019, -61.17, -88.952, 24.962, 62.488, -12.136]
  Call Extruder(8734.72433)
  MoveL 831 to (-5.78, 12.01, 40) mm, rotated rx -180 ry 0 rz 180 deg; joints [-157.997, -61.029, -89.461, 24.906, 62.826, -11.972]
  Call Extruder(8739.38797)
  MoveL 832 to (-8.31, 10.42, 40) mm, rotated rx -180 ry 0 rz 180 deg; joints [-158.08, -60.893, -89.96, 24.737, 63.138, -11.76]
  Call Extruder(8744.05216)
  MoveL 833 to (-10.42, 8.31, 40) mm, rotated rx 180 ry 0 rz 180 deg; joints [-158.266, -60.768, -90.424, 24.462, 63.409, -11.51]
  Call Extruder(8748.71578)
  MoveL 834 to (-12.01, 5.78, 40) mm, rotated rx 180 ry 0 rz -180 deg; joints [-158.549, -60.66, -90.83, 24.092, 63.625, -11.235]
  Call Extruder(8753.37935)
  MoveL 835 to (-13, 2.97, 40) mm, rotated rx -180 ry 0 rz -180 deg; joints [-158.913, -60.575, -91.156, 23.645, 63.774, -10.95]
  Call Extruder(8758.04331)
  MoveL 836 to (-13.33, 0, 40) mm, rotated rx 180 ry 0 rz 180 deg; joints [-159.341, -60.515, -91.385, 23.143, 63.85, -10.668]
  Call Extruder(8762.70726)
  MoveL 837 to (-12.99, -2.97, 40) mm, rotated rx 180 ry 0 rz -180 deg; joints [-159.811, -60.484, -91.506, 22.612, 63.846, -10.403]
  Call Extruder(8767.37083)
  MoveL 838 to (-12.01, -5.78, 40) mm, rotated rx -180 ry 0 rz 180 deg; joints [-160.294, -60.482, -91.511, 22.081, 63.764, -10.167]
  Call Extruder(8772.03446)
  MoveL 839 to (-10.42, -8.31, 40) mm, rotated rx 180 ry 0 rz 180 deg; joints [-160.766, -60.51, -91.402, 21.577, 63.606, -9.971]
  Call Extruder(8776.69865)
  MoveL 840 to (-8.31, -10.42, 40) mm, rotated rx 180 ry 0 rz 180 deg; joints [-161.2, -60.567, -91.183, 21.13, 63.381, -9.824]
  Call Extruder(8781.36227)
  MoveL 841 to (-5.78, -12.01, 40) mm, rotated rx 180 ry 0 rz 180 deg; joints [-161.572, -60.651, -90.866, 20.761, 63.099, -9.733]
  Call Extruder(8786.02584)
  MoveL 842 to (-2.97, -13, 40) mm, rotated rx -180 ry 0 rz 180 deg; joints [-161.863, -60.756, -90.468, 20.492, 62.776, -9.702]
  Call Extruder(8790.68979)
  MoveL 843 to (0, -13.33, 40) mm, rotated rx 180 ry 0 rz -180 deg; joints [-162.059, -60.88, -90.008, 20.335, 62.428, -9.734]
  Call Extruder(8792.60471)
  MoveL 844 to (1.22, -13.19, 40) mm, rotated rx -180 ry 0 rz 180 deg; joints [-162.097, -60.935, -89.805, 20.319, 62.283, -9.772]
  Set speed (130.0 mm/s)
  MoveL 845 to (1.22, -13.19, 45) mm, rotated rx 180 ry 0 rz 180 deg; joints [-162.097, -60.166, -90.226, 20.383, 61.957, -9.909]
  MoveL 846 to (-26.25, -4.54, 45) mm, rotated rx 180 ry 0 rz 180 deg; joints [-159.288, -59.156, -94.08, 22.951, 65.088, -10.114]
  Call Extruder(8794.83733)
  Set speed (60.0 mm/s)
  MoveL 847 to (-26.09, -5.96, 45) mm, rotated rx 180 ry 0 rz -180 deg; joints [-159.522, -59.141, -94.137, 22.69, 65.087, -9.989]
  Call Extruder(8804.20213)
  MoveL 848 to (-24.11, -11.61, 45) mm, rotated rx 180 ry 0 rz 180 deg; joints [-160.532, -59.139, -94.149, 21.59, 64.924, -9.521]
  Call Extruder(8813.56705)
  MoveL 849 to (-20.93, -16.69, 45) mm, rotated rx 180 ry 0 rz 180 deg; joints [-161.513, -59.194, -93.925, 20.548, 64.608, -9.132]
  Call Extruder(8822.93225)
  MoveL 850 to (-16.69, -20.93, 45) mm, rotated rx -180 ry 0 rz -180 deg; joints [-162.406, -59.305, -93.477, 19.625, 64.153, -8.836]
  Call Extruder(8832.29717)
  MoveL 851 to (-11.61, -24.12, 45) mm, rotated rx 180 ry 0 rz 180 deg; joints [-163.159, -59.469, -92.832, 18.874, 63.583, -8.648]
  Call Extruder(8841.66196)
  MoveL 852 to (-5.96, -26.09, 45) mm, rotated rx -180 ry 0 rz 180 deg; joints [-163.733, -59.68, -92.022, 18.335, 62.93, -8.576]
  Call Extruder(8851.02708)
  MoveL 853 to (0, -26.77, 45) mm, rotated rx 180 ry 0 rz 180 deg; joints [-164.103, -59.928, -91.092, 18.033, 62.227, -8.626]
  Call Extruder(8860.39217)
  MoveL 854 to (5.96, -26.09, 45) mm, rotated rx 180 ry 0 rz 180 deg; joints [-164.258, -60.204, -90.09, 17.98, 61.512, -8.799]
  Call Extruder(8869.75697)
  MoveL 855 to (11.61, -24.11, 45) mm, rotated rx 180 ry 0 rz 180 deg; joints [-164.201, -60.493, -89.066, 18.17, 60.823, -9.09]
  Call Extruder(8879.12188)
  MoveL 856 to (16.69, -20.93, 45) mm, rotated rx 180 ry 0 rz 180 deg; joints [-163.944, -60.782, -88.071, 18.587, 60.195, -9.489]
  Call Extruder(8888.48709)
  MoveL 857 to (20.93, -16.69, 45) mm, rotated rx 180 ry 0 rz 180 deg; joints [-163.508, -61.054, -87.155, 19.204, 59.659, -9.979]
  Call Extruder(8897.85201)
  MoveL 858 to (24.12, -11.61, 45) mm, rotated rx 180 ry 0 rz 180 deg; joints [-162.92, -61.294, -86.361, 19.986, 59.242, -10.537]
  Call Extruder(8907.21680)
  MoveL 859 to (26.09, -5.96, 45) mm, rotated rx -180 ry 0 rz -180 deg; joints [-162.209, -61.489, -85.726, 20.891, 58.964, -11.133]
  Call Extruder(8916.58191)
  MoveL 860 to (26.77, 0, 45) mm, rotated rx 180 ry 0 rz -180 deg; joints [-161.41, -61.627, -85.282, 21.873, 58.837, -11.736]
  Call Extruder(8925.94701)
  MoveL 861 to (26.09, 5.96, 45) mm, rotated rx -180 ry 0 rz 180 deg; joints [-160.556, -61.7, -85.049, 22.886, 58.867, -12.312]
  Call Extruder(8935.31181)
  MoveL 862 to (24.12, 11.61, 45) mm, rotated rx 180 ry 0 rz 180 deg; joints [-159.683, -61.704, -85.038, 23.882, 59.05, -12.828]
  Call Extruder(8944.67673)
  MoveL 863 to (20.93, 16.69, 45) mm, rotated rx 180 ry 0 rz 180 deg; joints [-158.826, -61.638, -85.249, 24.819, 59.375, -13.256]
  Call Extruder(8954.04193)
  MoveL 864 to (16.69, 20.93, 45) mm, rotated rx -180 ry 0 rz -180 deg; joints [-158.019, -61.506, -85.673, 25.655, 59.827, -13.572]
  Call Extruder(8963.40685)
  MoveL 865 to (11.61, 24.11, 45) mm, rotated rx 180 ry 0 rz 180 deg; joints [-157.299, -61.316, -86.29, 26.355, 60.381, -13.759]
  Call Extruder(8972.77165)
  MoveL 866 to (5.96, 26.09, 45) mm, rotated rx 180 ry 0 rz 180 deg; joints [-156.697, -61.08, -87.07, 26.889, 61.01, -13.807]
  Call Extruder(8982.13676)
  MoveL 867 to (0, 26.77, 45) mm, rotated rx -180 ry 0 rz 180 deg; joints [-156.245, -60.81, -87.976, 27.231, 61.685, -13.717]
  Call Extruder(8991.50186)
  MoveL 868 to (-5.96, 26.09, 45) mm, rotated rx -180 ry 0 rz 180 deg; joints [-155.969, -60.522, -88.965, 27.364, 62.373, -13.496]
  Call Extruder(9000.86665)
  MoveL 869 to (-11.61, 24.11, 45) mm, rotated rx -180 ry 0 rz 180 deg; joints [-155.891, -60.232, -89.988, 27.275, 63.042, -13.156]
  Call Extruder(9010.23157)
  MoveL 870 to (-16.69, 20.93, 45) mm, rotated rx 180 ry 0 rz -180 deg; joints [-156.025, -59.955, -90.995, 26.963, 63.661, -12.719]
  Call Extruder(9019.59678)
  MoveL 871 to (-20.93, 16.69, 45) mm, rotated rx 180 ry 0 rz 180 deg; joints [-156.374, -59.703, -91.934, 26.433, 64.2, -12.208]
  Call Extruder(9028.96169)
  MoveL 872 to (-24.11, 11.61, 45) mm, rotated rx -180 ry 0 rz 180 deg; joints [-156.928, -59.488, -92.758, 25.703, 64.632, -11.652]
  Call Extruder(9038.32649)
  MoveL 873 to (-26.09, 5.96, 45) mm, rotated rx -180 ry 0 rz -180 deg; joints [-157.665, -59.319, -93.422, 24.805, 64.934, -11.078]
  Call Extruder(9047.69160)
  MoveL 874 to (-26.77, 0, 45) mm, rotated rx 180 ry 0 rz 180 deg; joints [-158.546, -59.202, -93.89, 23.783, 65.09, -10.515]
  Call Extruder(9052.48033)
  MoveL 875 to (-26.42, -3.05, 45) mm, rotated rx -180 ry 0 rz -180 deg; joints [-159.044, -59.171, -94.018, 23.225, 65.089, -10.246]
  Set speed (130.0 mm/s)
  MoveL 876 to (-41.86, -6.3, 45) mm, rotated rx 180 ry 0 rz 180 deg; joints [-158.606, -58.579, -96.544, 23.357, 66.941, -9.601]
  Call Extruder(9057.47818)
  Set speed (60.0 mm/s)
  MoveL 877 to (-41.5, -9.47, 45) mm, rotated rx 180 ry 0 rz -180 deg; joints [-159.151, -58.551, -96.673, 22.755, 66.944, -9.329]
  Call Extruder(9072.37382)
  MoveL 878 to (-38.36, -18.47, 45) mm, rotated rx 180 ry 0 rz 180 deg; joints [-160.835, -58.546, -96.693, 20.943, 66.695, -8.61]
  Call Extruder(9087.26968)
  MoveL 879 to (-33.29, -26.54, 45) mm, rotated rx -180 ry 0 rz 180 deg; joints [-162.466, -58.627, -96.328, 19.226, 66.193, -8.013]
  Call Extruder(9102.16549)
  MoveL 880 to (-26.54, -33.28, 45) mm, rotated rx 180 ry 0 rz -180 deg; joints [-163.93, -58.792, -95.603, 17.716, 65.463, -7.557]
  Call Extruder(9117.06135)
  MoveL 881 to (-18.47, -38.36, 45) mm, rotated rx 180 ry 0 rz 180 deg; joints [-165.137, -59.039, -94.558, 16.505, 64.545, -7.257]
  Call Extruder(9131.95700)
  MoveL 882 to (-9.47, -41.5, 45) mm, rotated rx 180 ry 0 rz 180 deg; joints [-166.024, -59.361, -93.255, 15.657, 63.491, -7.131]
  Call Extruder(9146.85288)
  MoveL 883 to (0, -42.57, 45) mm, rotated rx 180 ry 0 rz 180 deg; joints [-166.562, -59.748, -91.765, 15.208, 62.361, -7.188]
  Call Extruder(9149.38031)
  MoveL 884 to (1.61, -42.39, 45) mm, rotated rx -180 ry 0 rz 180 deg; joints [-166.594, -59.819, -91.496, 15.2, 62.166, -7.23]
  Call Extruder(9161.74874)
  MoveL 885 to (9.47, -41.5, 45) mm, rotated rx 180 ry 0 rz 180 deg; joints [-166.745, -60.182, -90.167, 15.166, 61.215, -7.436]
  Call Extruder(9176.64441)
  MoveL 886 to (18.47, -38.36, 45) mm, rotated rx 180 ry 0 rz 180 deg; joints [-166.591, -60.645, -88.541, 15.513, 60.113, -7.875]
  Call Extruder(9191.54025)
  MoveL 887 to (26.54, -33.29, 45) mm, rotated rx 180 ry 0 rz 180 deg; joints [-166.133, -61.111, -86.966, 16.218, 59.112, -8.493]
  Call Extruder(9206.43607)
  MoveL 888 to (33.29, -26.54, 45) mm, rotated rx -180 ry 0 rz 180 deg; joints [-165.409, -61.554, -85.519, 17.23, 58.261, -9.266]
  Call Extruder(9221.33193)
  MoveL 889 to (38.36, -18.47, 45) mm, rotated rx 180 ry 0 rz 180 deg; joints [-164.468, -61.947, -84.267, 18.49, 57.603, -10.158]
  Call Extruder(9236.22758)
  MoveL 890 to (41.51, -9.47, 45) mm, rotated rx 180 ry 0 rz 180 deg; joints [-163.355, -62.268, -83.269, 19.931, 57.169, -11.122]
  Call Extruder(9251.12345)
  MoveL 891 to (42.57, 0, 45) mm, rotated rx 180 ry 0 rz 180 deg; joints [-162.12, -62.496, -82.57, 21.481, 56.977, -12.104]
  Call Extruder(9266.01932)
  MoveL 892 to (41.5, 9.47, 45) mm, rotated rx -180 ry 0 rz 180 deg; joints [-160.81, -62.617, -82.203, 23.065, 57.034, -13.045]
  Call Extruder(9280.91499)
  MoveL 893 to (38.36, 18.47, 45) mm, rotated rx 180 ry 0 rz 180 deg; joints [-159.475, -62.623, -82.186, 24.614, 57.335, -13.888]
  Call Extruder(9295.81083)
  MoveL 894 to (33.29, 26.54, 45) mm, rotated rx 180 ry 0 rz 180 deg; joints [-158.16, -62.513, -82.518, 26.062, 57.86, -14.584]
  Call Extruder(9310.70665)
  MoveL 895 to (26.54, 33.28, 45) mm, rotated rx 180 ry 0 rz 180 deg; joints [-156.916, -62.295, -83.185, 27.352, 58.58, -15.092]
  Call Extruder(9325.60250)
  MoveL 896 to (18.47, 38.36, 45) mm, rotated rx 180 ry 0 rz -180 deg; joints [-155.789, -61.983, -84.156, 28.435, 59.458, -15.386]
  Call Extruder(9340.49816)
  MoveL 897 to (9.47, 41.51, 45) mm, rotated rx 180 ry 0 rz 180 deg; joints [-154.828, -61.595, -85.385, 29.27, 60.451, -15.452]
  Call Extruder(9355.39403)
  MoveL 898 to (0, 42.57, 45) mm, rotated rx 180 ry 0 rz -180 deg; joints [-154.081, -61.156, -86.816, 29.823, 61.511, -15.292]
  Call Extruder(9370.28991)
  MoveL 899 to (-9.47, 41.51, 45) mm, rotated rx -180 ry 0 rz 180 deg; joints [-153.594, -60.692, -88.381, 30.064, 62.591, -14.92]
  Call Extruder(9385.18556)
  MoveL 900 to (-18.47, 38.36, 45) mm, rotated rx 180 ry 0 rz -180 deg; joints [-153.408, -60.228, -90.005, 29.971, 63.643, -14.36]
  Call Extruder(9400.08141)
  MoveL 901 to (-26.54, 33.29, 45) mm, rotated rx -180 ry 0 rz -180 deg; joints [-153.557, -59.789, -91.61, 29.53, 64.62, -13.647]
  Call Extruder(9414.97723)
  MoveL 902 to (-33.29, 26.54, 45) mm, rotated rx 180 ry 0 rz 180 deg; joints [-154.059, -59.397, -93.115, 28.739, 65.476, -12.823]
  Call Extruder(9429.87308)
  MoveL 903 to (-38.36, 18.47, 45) mm, rotated rx 180 ry 0 rz 180 deg; joints [-154.913, -59.068, -94.439, 27.613, 66.171, -11.933]
  Call Extruder(9444.76874)
  MoveL 904 to (-41.51, 9.47, 45) mm, rotated rx 180 ry 0 rz 180 deg; joints [-156.091, -58.813, -95.512, 26.193, 66.667, -11.025]
  Call Extruder(9459.66461)
  MoveL 905 to (-42.57, 0, 45) mm, rotated rx 180 ry 0 rz -180 deg; joints [-157.533, -58.64, -96.272, 24.542, 66.932, -10.144]
  Call Extruder(9467.21888)
  MoveL 906 to (-42.03, -4.8, 45) mm, rotated rx -180 ry 0 rz 180 deg; joints [-158.35, -58.593, -96.481, 23.639, 66.939, -9.729]
  Set speed (130.0 mm/s)
  MoveL 907 to (-54.1, -7.67, 45) mm, rotated rx -180 ry 0 rz 180 deg; joints [-158.024, -58.18, -98.43, 23.734, 68.399, -9.194]
  Call Extruder(9471.29152)
  Set speed (30.0 mm/s)
  MoveL 908 to (-53.59, -12.23, 45) mm, rotated rx 180 ry 0 rz -180 deg; joints [-158.835, -58.142, -98.619, 22.848, 68.41, -8.813]
  Call Extruder(9482.22165)
  MoveL 909 to (-49.53, -23.85, 45) mm, rotated rx -180 ry 0 rz 180 deg; joints [-161.095, -58.137, -98.644, 20.438, 68.101, -7.913]
  Call Extruder(9493.15193)
  MoveL 910 to (-42.98, -34.27, 45) mm, rotated rx 180 ry 0 rz 180 deg; joints [-163.275, -58.234, -98.164, 18.155, 67.453, -7.167]
  Call Extruder(9504.08205)
  MoveL 911 to (-34.27, -42.98, 45) mm, rotated rx -180 ry 0 rz 180 deg; joints [-165.21, -58.434, -97.211, 16.162, 66.501, -6.592]
  Call Extruder(9515.01234)
  MoveL 912 to (-23.85, -49.53, 45) mm, rotated rx -180 ry 0 rz -180 deg; joints [-166.774, -58.737, -95.845, 14.586, 65.302, -6.205]
  Call Extruder(9525.94247)
  MoveL 913 to (-12.23, -53.59, 45) mm, rotated rx -180 ry 0 rz 180 deg; joints [-167.889, -59.139, -94.147, 13.508, 63.926, -6.027]
  Call Extruder(9536.87269)
  MoveL 914 to (0, -54.97, 45) mm, rotated rx 180 ry 0 rz 180 deg; joints [-168.526, -59.63, -92.213, 12.965, 62.453, -6.077]
  Call Extruder(9539.54151)
  MoveL 915 to (2.99, -54.63, 45) mm, rotated rx 180 ry 0 rz 180 deg; joints [-168.569, -59.762, -91.712, 12.96, 62.089, -6.148]
  Call Extruder(9547.80291)
  MoveL 916 to (12.23, -53.59, 45) mm, rotated rx -180 ry 0 rz 180 deg; joints [-168.697, -60.188, -90.145, 12.954, 60.965, -6.37]
  Call Extruder(9558.73305)
  MoveL 917 to (23.85, -49.53, 45) mm, rotated rx 180 ry 0 rz 180 deg; joints [-168.436, -60.789, -88.049, 13.447, 59.538, -6.912]
  Call Extruder(9569.66333)
  MoveL 918 to (34.27, -42.98, 45) mm, rotated rx 180 ry 0 rz 180 deg; joints [-167.797, -61.397, -86.025, 14.394, 58.245, -7.692]
  Call Extruder(9580.59345)
  MoveL 919 to (42.98, -34.27, 45) mm, rotated rx 180 ry 0 rz 180 deg; joints [-166.837, -61.979, -84.166, 15.727, 57.15, -8.685]
  Call Extruder(9591.52374)
  MoveL 920 to (49.53, -23.85, 45) mm, rotated rx -180 ry 0 rz 180 deg; joints [-165.618, -62.499, -82.56, 17.37, 56.305, -9.845]
  Call Extruder(9602.45387)
  MoveL 921 to (53.59, -12.23, 45) mm, rotated rx -180 ry 0 rz -180 deg; joints [-164.2, -62.924, -81.28, 19.232, 55.75, -11.108]
  Call Extruder(9613.38409)
  MoveL 922 to (54.97, 0, 45) mm, rotated rx 180 ry 0 rz 180 deg; joints [-162.641, -63.226, -80.384, 21.223, 55.511, -12.401]
  Call Extruder(9624.31431)
  MoveL 923 to (53.59, 12.23, 45) mm, rotated rx -180 ry 0 rz 180 deg; joints [-160.996, -63.387, -79.914, 23.246, 55.595, -13.643]
  Call Extruder(9635.24446)
  MoveL 924 to (49.53, 23.85, 45) mm, rotated rx 180 ry 0 rz -180 deg; joints [-159.322, -63.394, -79.891, 25.212, 55.992, -14.753]
  Call Extruder(9646.17473)
  MoveL 925 to (42.98, 34.27, 45) mm, rotated rx -180 ry 0 rz 180 deg; joints [-157.673, -63.249, -80.318, 27.042, 56.677, -15.665]
  Call Extruder(9657.10486)
  MoveL 926 to (34.27, 42.98, 45) mm, rotated rx 180 ry 0 rz 180 deg; joints [-156.102, -62.96, -81.173, 28.669, 57.61, -16.325]
  Call Extruder(9668.03513)
  MoveL 927 to (23.85, 49.52, 45) mm, rotated rx 180 ry 0 rz 180 deg; joints [-154.667, -62.546, -82.418, 30.035, 58.742, -16.699]
  Call Extruder(9678.96528)
  MoveL 928 to (12.23, 53.59, 45) mm, rotated rx 180 ry 0 rz -180 deg; joints [-153.426, -62.034, -83.994, 31.096, 60.017, -16.774]
  Call Extruder(9689.89550)
  MoveL 929 to (0, 54.97, 45) mm, rotated rx 180 ry 0 rz 180 deg; joints [-152.438, -61.457, -85.831, 31.813, 61.375, -16.551]
  Call Extruder(9700.82572)
  MoveL 930 to (-12.23, 53.59, 45) mm, rotated rx 180 ry 0 rz 180 deg; joints [-151.764, -60.849, -87.844, 32.15, 62.755, -16.052]
  Call Extruder(9711.75585)
  MoveL 931 to (-23.85, 49.52, 45) mm, rotated rx -180 ry 0 rz 180 deg; joints [-151.463, -60.247, -89.937, 32.077, 64.099, -15.311]
  Call Extruder(9722.68614)
  MoveL 932 to (-34.27, 42.98, 45) mm, rotated rx 180 ry 0 rz 180 deg; joints [-151.589, -59.682, -92.012, 31.567, 65.35, -14.373]
  Call Extruder(9733.61626)
  MoveL 933 to (-42.98, 34.27, 45) mm, rotated rx 180 ry 0 rz -180 deg; joints [-152.179, -59.184, -93.964, 30.603, 66.454, -13.294]
  Call Extruder(9744.54654)
  MoveL 934 to (-49.52, 23.85, 45) mm, rotated rx 180 ry 0 rz 180 deg; joints [-153.248, -58.772, -95.69, 29.191, 67.359, -12.138]
  Call Extruder(9755.47668)
  MoveL 935 to (-53.59, 12.23, 45) mm, rotated rx 180 ry 0 rz -180 deg; joints [-154.769, -58.459, -97.093, 27.368, 68.014, -10.968]
  Call Extruder(9766.40690)
  MoveL 936 to (-54.97, 0, 45) mm, rotated rx 180 ry 0 rz -180 deg; joints [-156.673, -58.249, -98.09, 25.212, 68.376, -9.843]
  Call Extruder(9771.93251)
  MoveL 937 to (-54.27, -6.18, 45) mm, rotated rx 180 ry 0 rz 180 deg; joints [-157.76, -58.193, -98.367, 24.022, 68.395, -9.319]
  Set speed (130.0 mm/s)
  MoveL 938 to (-49.9, -9.51, 45) mm, rotated rx 180 ry 0 rz 180 deg; joints [-158.616, -58.284, -97.921, 23.168, 67.933, -9.134]
  MoveL 939 to (2.97, -12.99, 45) mm, rotated rx -180 ry 0 rz -180 deg; joints [-162.152, -60.248, -89.932, 20.361, 61.749, -9.963]
  Call Extruder(9776.59609)
  Set speed (80.0 mm/s)
  MoveL 940 to (5.78, -12.01, 45) mm, rotated rx 180 ry 0 rz -180 deg; joints [-162.141, -60.392, -89.422, 20.443, 61.407, -10.115]
  Call Extruder(9781.25971)
  MoveL 941 to (8.31, -10.42, 45) mm, rotated rx 180 ry 0 rz -180 deg; joints [-162.027, -60.534, -88.925, 20.639, 61.095, -10.318]
  Call Extruder(9785.92390)
  MoveL 942 to (10.42, -8.31, 45) mm, rotated rx -180 ry 0 rz 180 deg; joints [-161.819, -60.667, -88.466, 20.937, 60.828, -10.564]
  Call Extruder(9790.58754)
  MoveL 943 to (12.01, -5.78, 45) mm, rotated rx 180 ry 0 rz 180 deg; joints [-161.529, -60.783, -88.067, 21.322, 60.618, -10.841]
  Call Extruder(9795.25110)
  MoveL 944 to (12.99, -2.97, 45) mm, rotated rx 180 ry 0 rz -180 deg; joints [-161.171, -60.877, -87.748, 21.772, 60.477, -11.134]
  Call Extruder(9799.91505)
  MoveL 945 to (13.33, 0, 45) mm, rotated rx 180 ry 0 rz 180 deg; joints [-160.763, -60.944, -87.524, 22.265, 60.411, -11.429]
  Call Extruder(9804.57901)
  MoveL 946 to (12.99, 2.97, 45) mm, rotated rx -180 ry 0 rz 180 deg; joints [-160.324, -60.979, -87.407, 22.777, 60.423, -11.709]
  Call Extruder(9809.24258)
  MoveL 947 to (12.01, 5.78, 45) mm, rotated rx 180 ry 0 rz -180 deg; joints [-159.874, -60.98, -87.401, 23.285, 60.512, -11.961]
  Call Extruder(9813.90620)
  MoveL 948 to (10.42, 8.31, 45) mm, rotated rx -180 ry 0 rz 180 deg; joints [-159.432, -60.949, -87.508, 23.763, 60.672, -12.17]
  Call Extruder(9818.57039)
  MoveL 949 to (8.31, 10.42, 45) mm, rotated rx 180 ry 0 rz 180 deg; joints [-159.021, -60.885, -87.721, 24.19, 60.897, -12.325]
  Call Extruder(9823.23402)
  MoveL 950 to (5.78, 12.01, 45) mm, rotated rx 180 ry 0 rz 180 deg; joints [-158.657, -60.794, -88.031, 24.546, 61.174, -12.418]
  Call Extruder(9827.89760)
  MoveL 951 to (2.97, 13, 45) mm, rotated rx 180 ry 0 rz 180 deg; joints [-158.359, -60.679, -88.423, 24.814, 61.49, -12.445]
  Call Extruder(9832.56155)
  MoveL 952 to (0, 13.33, 45) mm, rotated rx 180 ry 0 rz 180 deg; joints [-158.143, -60.548, -88.878, 24.981, 61.829, -12.405]
  Call Extruder(9837.22550)
  MoveL 953 to (-2.97, 12.99, 45) mm, rotated rx 180 ry 0 rz 180 deg; joints [-158.019, -60.406, -89.372, 25.039, 62.176, -12.3]
  Call Extruder(9841.88907)
  MoveL 954 to (-5.78, 12.01, 45) mm, rotated rx 180 ry 0 rz 180 deg; joints [-157.997, -60.262, -89.882, 24.982, 62.512, -12.137]
  Call Extruder(9846.55270)
  MoveL 955 to (-8.31, 10.42, 45) mm, rotated rx -180 ry 0 rz -180 deg; joints [-158.08, -60.123, -90.382, 24.812, 62.822, -11.924]
  Call Extruder(9851.21689)
  MoveL 956 to (-10.42, 8.31, 45) mm, rotated rx 180 ry 0 rz 180 deg; joints [-158.266, -59.995, -90.847, 24.535, 63.09, -11.673]
  Call Extruder(9855.88051)
  MoveL 957 to (-12.01, 5.78, 45) mm, rotated rx 180 ry 0 rz 180 deg; joints [-158.549, -59.885, -91.253, 24.164, 63.303, -11.396]
  Call Extruder(9860.54408)
  MoveL 958 to (-12.99, 2.97, 45) mm, rotated rx 180 ry 0 rz -180 deg; joints [-158.913, -59.797, -91.58, 23.715, 63.451, -11.109]
  Call Extruder(9865.20804)
  MoveL 959 to (-13.33, 0, 45) mm, rotated rx 180 ry 0 rz 180 deg; joints [-159.341, -59.736, -91.809, 23.212, 63.524, -10.824]
  Call Extruder(9869.87199)
  MoveL 960 to (-12.99, -2.97, 45) mm, rotated rx 180 ry 0 rz 180 deg; joints [-159.811, -59.704, -91.93, 22.68, 63.519, -10.556]
  Call Extruder(9874.53556)
  MoveL 961 to (-12.01, -5.78, 45) mm, rotated rx 180 ry 0 rz 180 deg; joints [-160.294, -59.702, -91.936, 22.147, 63.435, -10.316]
  Call Extruder(9879.19919)
  MoveL 962 to (-10.42, -8.31, 45) mm, rotated rx 180 ry 0 rz 180 deg; joints [-160.766, -59.731, -91.826, 21.643, 63.276, -10.117]
  Call Extruder(9883.86338)
  MoveL 963 to (-8.31, -10.42, 45) mm, rotated rx 180 ry 0 rz 180 deg; joints [-161.2, -59.79, -91.607, 21.194, 63.051, -9.967]
  Call Extruder(9888.52701)
  MoveL 964 to (-5.78, -12.01, 45) mm, rotated rx 180 ry 0 rz 180 deg; joints [-161.572, -59.875, -91.29, 20.825, 62.77, -9.873]
  Call Extruder(9893.19057)
  MoveL 965 to (-2.97, -13, 45) mm, rotated rx 180 ry 0 rz 180 deg; joints [-161.863, -59.983, -90.89, 20.556, 62.448, -9.84]
  Call Extruder(9897.85454)
  MoveL 966 to (0, -13.33, 45) mm, rotated rx 180 ry 0 rz -180 deg; joints [-162.059, -60.109, -90.43, 20.399, 62.102, -9.871]
  Call Extruder(9902.51848)
  MoveL 967 to (2.97, -12.99, 45) mm, rotated rx -180 ry 0 rz -180 deg; joints [-162.152, -60.248, -89.932, 20.361, 61.749, -9.963]
  Set speed (130.0 mm/s)
  MoveL 968 to (2.97, -12.99, 50) mm, rotated rx 180 ry 0 rz -180 deg; joints [-162.152, -59.481, -90.344, 20.428, 61.416, -10.104]
  MoveL 969 to (-26.25, -4.54, 50) mm, rotated rx 180 ry 0 rz 180 deg; joints [-159.288, -58.361, -94.5, 23.02, 64.744, -10.275]
  Call Extruder(9904.75110)
  Set speed (60.0 mm/s)
  MoveL 970 to (-26.09, -5.96, 50) mm, rotated rx 180 ry 0 rz 180 deg; joints [-159.522, -58.347, -94.557, 22.758, 64.742, -10.148]
  Call Extruder(9914.11589)
  MoveL 971 to (-24.12, -11.61, 50) mm, rotated rx -180 ry 0 rz 180 deg; joints [-160.532, -58.344, -94.569, 21.656, 64.576, -9.674]
  Call Extruder(9923.48081)
  MoveL 972 to (-20.93, -16.69, 50) mm, rotated rx -180 ry 0 rz 180 deg; joints [-161.513, -58.401, -94.344, 20.611, 64.258, -9.277]
  Call Extruder(9932.84602)
  MoveL 973 to (-16.69, -20.93, 50) mm, rotated rx 180 ry 0 rz 180 deg; joints [-162.406, -58.515, -93.896, 19.686, 63.803, -8.975]
  Call Extruder(9942.21094)
  MoveL 974 to (-11.61, -24.12, 50) mm, rotated rx 180 ry 0 rz 180 deg; joints [-163.159, -58.683, -93.249, 18.934, 63.235, -8.782]
  Call Extruder(9951.57573)
  MoveL 975 to (-5.96, -26.09, 50) mm, rotated rx 180 ry 0 rz 180 deg; joints [-163.733, -58.899, -92.438, 18.394, 62.584, -8.706]
  Call Extruder(9960.94082)
  MoveL 976 to (0, -26.77, 50) mm, rotated rx 180 ry 0 rz 180 deg; joints [-164.103, -59.154, -91.506, 18.093, 61.884, -8.753]
  Call Extruder(9970.30594)
  MoveL 977 to (5.96, -26.09, 50) mm, rotated rx 180 ry 0 rz 180 deg; joints [-164.258, -59.436, -90.502, 18.04, 61.174, -8.924]
  Call Extruder(9979.67074)
  MoveL 978 to (11.61, -24.11, 50) mm, rotated rx 180 ry 0 rz 180 deg; joints [-164.201, -59.731, -89.477, 18.231, 60.489, -9.216]
  Call Extruder(9989.03565)
  MoveL 979 to (16.69, -20.93, 50) mm, rotated rx 180 ry 0 rz 180 deg; joints [-163.944, -60.026, -88.481, 18.651, 59.866, -9.617]
  Call Extruder(9998.40086)
  MoveL 980 to (20.93, -16.69, 50) mm, rotated rx -180 ry 0 rz 180 deg; joints [-163.508, -60.303, -87.563, 19.271, 59.335, -10.111]
  Call Extruder(10007.76578)
  MoveL 981 to (24.12, -11.61, 50) mm, rotated rx 180 ry 0 rz 180 deg; joints [-162.92, -60.547, -86.768, 20.056, 58.922, -10.672]
  Call Extruder(10017.13057)
  MoveL 982 to (26.09, -5.96, 50) mm, rotated rx 180 ry 0 rz -180 deg; joints [-162.209, -60.746, -86.133, 20.964, 58.649, -11.274]
  Call Extruder(10026.49568)
  MoveL 983 to (26.77, 0, 50) mm, rotated rx 180 ry 0 rz -180 deg; joints [-161.41, -60.886, -85.688, 21.949, 58.526, -11.882]
  Call Extruder(10035.86078)
  MoveL 984 to (26.09, 5.96, 50) mm, rotated rx -180 ry 0 rz 180 deg; joints [-160.556, -60.96, -85.455, 22.965, 58.559, -12.464]
  Call Extruder(10045.22559)
  MoveL 985 to (24.11, 11.61, 50) mm, rotated rx 180 ry 0 rz 180 deg; joints [-159.683, -60.964, -85.443, 23.964, 58.744, -12.987]
  Call Extruder(10054.59050)
  MoveL 986 to (20.93, 16.69, 50) mm, rotated rx -180 ry 0 rz 180 deg; joints [-158.826, -60.897, -85.655, 24.903, 59.071, -13.42]
  Call Extruder(10063.95571)
  MoveL 987 to (16.69, 20.93, 50) mm, rotated rx -180 ry 0 rz 180 deg; joints [-158.019, -60.762, -86.08, 25.741, 59.523, -13.741]
  Call Extruder(10073.32062)
  MoveL 988 to (11.61, 24.11, 50) mm, rotated rx -180 ry 0 rz 180 deg; joints [-157.299, -60.569, -86.697, 26.442, 60.077, -13.933]
  Call Extruder(10082.68542)
  MoveL 989 to (5.96, 26.09, 50) mm, rotated rx 180 ry 0 rz 180 deg; joints [-156.697, -60.329, -87.478, 26.975, 60.704, -13.985]
  Call Extruder(10092.05053)
  MoveL 990 to (0, 26.77, 50) mm, rotated rx -180 ry 0 rz 180 deg; joints [-156.245, -60.054, -88.385, 27.317, 61.376, -13.898]
  Call Extruder(10101.41563)
  MoveL 991 to (-5.96, 26.09, 50) mm, rotated rx -180 ry 0 rz 180 deg; joints [-155.969, -59.761, -89.376, 27.449, 62.061, -13.678]
  Call Extruder(10110.78042)
  MoveL 992 to (-11.61, 24.12, 50) mm, rotated rx -180 ry 0 rz 180 deg; joints [-155.891, -59.465, -90.4, 27.359, 62.726, -13.339]
  Call Extruder(10120.14534)
  MoveL 993 to (-16.69, 20.93, 50) mm, rotated rx -180 ry 0 rz -180 deg; joints [-156.025, -59.181, -91.409, 27.044, 63.34, -12.901]
  Call Extruder(10129.51055)
  MoveL 994 to (-20.93, 16.69, 50) mm, rotated rx 180 ry 0 rz 180 deg; joints [-156.374, -58.923, -92.35, 26.512, 63.874, -12.389]
  Call Extruder(10138.87546)
  MoveL 995 to (-24.12, 11.61, 50) mm, rotated rx -180 ry 0 rz 180 deg; joints [-156.928, -58.703, -93.175, 25.779, 64.301, -11.829]
  Call Extruder(10148.24026)
  MoveL 996 to (-26.09, 5.96, 50) mm, rotated rx 180 ry 0 rz -180 deg; joints [-157.665, -58.529, -93.84, 24.879, 64.598, -11.251]
  Call Extruder(10157.60537)
  MoveL 997 to (-26.77, 0, 50) mm, rotated rx -180 ry 0 rz 180 deg; joints [-158.546, -58.409, -94.31, 23.853, 64.748, -10.682]
  Call Extruder(10162.39410)
  MoveL 998 to (-26.42, -3.05, 50) mm, rotated rx 180 ry 0 rz -180 deg; joints [-159.044, -58.377, -94.438, 23.294, 64.745, -10.409]
  Set speed (130.0 mm/s)
  MoveL 999 to (-41.86, -6.3, 50) mm, rotated rx -180 ry 0 rz -180 deg; joints [-158.606, -57.768, -96.969, 23.423, 66.586, -9.767]
  Call Extruder(10167.39195)
  Set speed (60.0 mm/s)
  MoveL 1000 to (-41.5, -9.47, 50) mm, rotated rx 180 ry 0 rz 180 deg; joints [-159.151, -57.738, -97.1, 22.82, 66.588, -9.491]
  Call Extruder(10182.28759)
  MoveL 1001 to (-38.36, -18.47, 50) mm, rotated rx 180 ry 0 rz 180 deg; joints [-160.835, -57.733, -97.119, 21.003, 66.334, -8.761]
  Call Extruder(10197.18345)
  MoveL 1002 to (-33.28, -26.54, 50) mm, rotated rx 180 ry 0 rz 180 deg; joints [-162.466, -57.817, -96.754, 19.283, 65.83, -8.152]
  Call Extruder(10212.07926)
  MoveL 1003 to (-26.54, -33.28, 50) mm, rotated rx 180 ry 0 rz -180 deg; joints [-163.93, -57.988, -96.026, 17.769, 65.1, -7.685]
  Call Extruder(10226.97512)
  MoveL 1004 to (-18.47, -38.36, 50) mm, rotated rx 180 ry 0 rz 180 deg; joints [-165.137, -58.242, -94.979, 16.556, 64.184, -7.376]
  Call Extruder(10241.87077)
  MoveL 1005 to (-9.47, -41.5, 50) mm, rotated rx 180 ry 0 rz -180 deg; joints [-166.024, -58.573, -93.673, 15.708, 63.135, -7.243]
  Call Extruder(10256.76664)
  MoveL 1006 to (0, -42.57, 50) mm, rotated rx 180 ry 0 rz 180 deg; joints [-166.562, -58.969, -92.181, 15.259, 62.01, -7.296]
  Call Extruder(10259.95013)
  MoveL 1007 to (2.03, -42.34, 50) mm, rotated rx 180 ry 0 rz 180 deg; joints [-166.602, -59.062, -91.84, 15.249, 61.766, -7.348]
  Call Extruder(10271.66252)
  MoveL 1008 to (9.47, -41.51, 50) mm, rotated rx 180 ry 0 rz 180 deg; joints [-166.745, -59.414, -90.579, 15.217, 60.871, -7.543]
  Call Extruder(10286.55818)
  MoveL 1009 to (18.47, -38.36, 50) mm, rotated rx -180 ry 0 rz 180 deg; joints [-166.591, -59.886, -88.95, 15.568, 59.776, -7.983]
  Call Extruder(10301.45402)
  MoveL 1010 to (26.54, -33.29, 50) mm, rotated rx -180 ry 0 rz 180 deg; joints [-166.133, -60.36, -87.374, 16.275, 58.783, -8.604]
  Call Extruder(10316.34984)
  MoveL 1011 to (33.29, -26.54, 50) mm, rotated rx 180 ry 0 rz 180 deg; joints [-165.409, -60.811, -85.925, 17.292, 57.94, -9.383]
  Call Extruder(10331.24570)
  MoveL 1012 to (38.36, -18.47, 50) mm, rotated rx -180 ry 0 rz 180 deg; joints [-164.468, -61.211, -84.672, 18.557, 57.289, -10.283]
  Call Extruder(10346.14135)
  MoveL 1013 to (41.5, -9.47, 50) mm, rotated rx -180 ry 0 rz 180 deg; joints [-163.355, -61.537, -83.673, 20.004, 56.862, -11.255]
  Call Extruder(10361.03722)
  MoveL 1014 to (42.57, 0, 50) mm, rotated rx 180 ry 0 rz 180 deg; joints [-162.12, -61.768, -82.974, 21.558, 56.675, -12.246]
  Call Extruder(10375.93309)
  MoveL 1015 to (41.51, 9.47, 50) mm, rotated rx -180 ry 0 rz 180 deg; joints [-160.81, -61.891, -82.607, 23.147, 56.738, -13.196]
  Call Extruder(10390.82876)
  MoveL 1016 to (38.36, 18.47, 50) mm, rotated rx 180 ry 0 rz 180 deg; joints [-159.475, -61.896, -82.589, 24.7, 57.042, -14.049]
  Call Extruder(10405.72460)
  MoveL 1017 to (33.29, 26.54, 50) mm, rotated rx -180 ry 0 rz 180 deg; joints [-158.16, -61.785, -82.922, 26.152, 57.569, -14.753]
  Call Extruder(10420.62042)
  MoveL 1018 to (26.54, 33.28, 50) mm, rotated rx 180 ry 0 rz 180 deg; joints [-156.916, -61.564, -83.589, 27.444, 58.29, -15.268]
  Call Extruder(10435.51627)
  MoveL 1019 to (18.47, 38.36, 50) mm, rotated rx -180 ry 0 rz -180 deg; joints [-155.789, -61.247, -84.561, 28.529, 59.167, -15.569]
  Call Extruder(10450.41193)
  MoveL 1020 to (9.47, 41.51, 50) mm, rotated rx 180 ry 0 rz 180 deg; joints [-154.828, -60.853, -85.791, 29.364, 60.158, -15.641]
  Call Extruder(10465.30781)
  MoveL 1021 to (0, 42.57, 50) mm, rotated rx 180 ry 0 rz 180 deg; joints [-154.081, -60.407, -87.224, 29.916, 61.215, -15.486]
  Call Extruder(10480.20368)
  MoveL 1022 to (-9.47, 41.51, 50) mm, rotated rx 180 ry 0 rz 180 deg; joints [-153.594, -59.933, -88.79, 30.155, 62.29, -15.117]
  Call Extruder(10495.09933)
  MoveL 1023 to (-18.47, 38.36, 50) mm, rotated rx 180 ry 0 rz 180 deg; joints [-153.408, -59.46, -90.418, 30.06, 63.335, -14.559]
  Call Extruder(10509.99518)
  MoveL 1024 to (-26.54, 33.29, 50) mm, rotated rx 180 ry 0 rz -180 deg; joints [-153.557, -59.011, -92.025, 29.615, 64.304, -13.846]
  Call Extruder(10524.89100)
  MoveL 1025 to (-33.28, 26.54, 50) mm, rotated rx 180 ry 0 rz 180 deg; joints [-154.059, -58.609, -93.533, 28.821, 65.152, -13.018]
  Call Extruder(10539.78685)
  MoveL 1026 to (-38.36, 18.47, 50) mm, rotated rx 180 ry 0 rz -180 deg; joints [-154.913, -58.271, -94.86, 27.691, 65.838, -12.124]
  Call Extruder(10554.68250)
  MoveL 1027 to (-41.5, 9.47, 50) mm, rotated rx 180 ry 0 rz -180 deg; joints [-156.091, -58.009, -95.936, 26.266, 66.325, -11.208]
  Call Extruder(10569.57838)
  MoveL 1028 to (-42.57, 0, 50) mm, rotated rx -180 ry 0 rz -180 deg; joints [-157.533, -57.83, -96.697, 24.611, 66.582, -10.318]
  Call Extruder(10577.13266)
  MoveL 1029 to (-42.03, -4.8, 50) mm, rotated rx 180 ry 0 rz -180 deg; joints [-158.35, -57.782, -96.907, 23.705, 66.586, -9.897]
  Set speed (130.0 mm/s)
  MoveL 1030 to (-54.1, -7.67, 50) mm, rotated rx 180 ry 0 rz 180 deg; joints [-158.024, -57.354, -98.861, 23.797, 68.038, -9.366]
  Call Extruder(10581.20529)
  Set speed (30.0 mm/s)
  MoveL 1031 to (-53.59, -12.23, 50) mm, rotated rx 180 ry 0 rz 180 deg; joints [-158.835, -57.315, -99.05, 22.91, 68.046, -8.979]
  Call Extruder(10592.13542)
  MoveL 1032 to (-49.52, -23.85, 50) mm, rotated rx 180 ry 0 rz -180 deg; joints [-161.095, -57.309, -99.076, 20.494, 67.729, -8.062]
  Call Extruder(10603.06570)
  MoveL 1033 to (-42.98, -34.27, 50) mm, rotated rx 180 ry 0 rz 180 deg; joints [-163.275, -57.41, -98.595, 18.207, 67.079, -7.3]
  Call Extruder(10613.99582)
  MoveL 1034 to (-34.27, -42.98, 50) mm, rotated rx 180 ry 0 rz 180 deg; joints [-165.21, -57.617, -97.639, 16.21, 66.128, -6.71]
  Call Extruder(10624.92611)
  MoveL 1035 to (-23.85, -49.53, 50) mm, rotated rx 180 ry 0 rz -180 deg; joints [-166.774, -57.93, -96.269, 14.631, 64.932, -6.312]
  Call Extruder(10635.85624)
  MoveL 1036 to (-12.23, -53.59, 50) mm, rotated rx -180 ry 0 rz 180 deg; joints [-167.889, -58.344, -94.567, 13.551, 63.562, -6.125]
  Call Extruder(10646.78646)
  MoveL 1037 to (0, -54.97, 50) mm, rotated rx -180 ry 0 rz 180 deg; joints [-168.526, -58.848, -92.629, 13.008, 62.097, -6.17]
  Call Extruder(10649.82812)
  MoveL 1038 to (3.4, -54.59, 50) mm, rotated rx -180 ry 0 rz 180 deg; joints [-168.575, -59.003, -92.057, 13.003, 61.685, -6.251]
  Call Extruder(10657.71668)
  MoveL 1039 to (12.23, -53.59, 50) mm, rotated rx -180 ry 0 rz 180 deg; joints [-168.697, -59.42, -90.558, 12.999, 60.618, -6.462]
  Call Extruder(10668.64683)
  MoveL 1040 to (23.85, -49.53, 50) mm, rotated rx 180 ry 0 rz 180 deg; joints [-168.436, -60.032, -88.458, 13.495, 59.201, -7.006]
  Call Extruder(10679.57711)
  MoveL 1041 to (34.27, -42.98, 50) mm, rotated rx -180 ry 0 rz 180 deg; joints [-167.797, -60.652, -86.431, 14.446, 57.918, -7.791]
  Call Extruder(10690.50723)
  MoveL 1042 to (42.98, -34.27, 50) mm, rotated rx -180 ry 0 rz 180 deg; joints [-166.837, -61.244, -84.571, 15.786, 56.831, -8.792]
  Call Extruder(10701.43751)
  MoveL 1043 to (49.52, -23.85, 50) mm, rotated rx -180 ry 0 rz 180 deg; joints [-165.618, -61.771, -82.964, 17.435, 55.995, -9.961]
  Call Extruder(10712.36764)
  MoveL 1044 to (53.59, -12.23, 50) mm, rotated rx -180 ry 0 rz -180 deg; joints [-164.2, -62.202, -81.683, 19.304, 55.449, -11.236]
  Call Extruder(10723.29786)
  MoveL 1045 to (54.97, 0, 50) mm, rotated rx -180 ry 0 rz 180 deg; joints [-162.641, -62.508, -80.787, 21.302, 55.217, -12.54]
  Call Extruder(10734.22808)
  MoveL 1046 to (53.59, 12.23, 50) mm, rotated rx 180 ry 0 rz 180 deg; joints [-160.996, -62.671, -80.316, 23.331, 55.307, -13.793]
  Call Extruder(10745.15823)
  MoveL 1047 to (49.52, 23.85, 50) mm, rotated rx -180 ry 0 rz -180 deg; joints [-159.322, -62.679, -80.294, 25.303, 55.708, -14.915]
  Call Extruder(10756.08850)
  MoveL 1048 to (42.98, 34.27, 50) mm, rotated rx -180 ry 0 rz 180 deg; joints [-157.673, -62.531, -80.72, 27.137, 56.396, -15.837]
  Call Extruder(10767.01863)
  MoveL 1049 to (34.27, 42.98, 50) mm, rotated rx 180 ry 0 rz 180 deg; joints [-156.102, -62.238, -81.576, 28.766, 57.331, -16.507]
  Call Extruder(10777.94890)
  MoveL 1050 to (23.85, 49.52, 50) mm, rotated rx -180 ry 0 rz -180 deg; joints [-154.667, -61.819, -82.821, 30.134, 58.462, -16.889]
  Call Extruder(10788.87905)
  MoveL 1051 to (12.23, 53.59, 50) mm, rotated rx 180 ry 0 rz 180 deg; joints [-153.426, -61.3, -84.399, 31.195, 59.734, -16.971]
  Call Extruder(10799.80927)
  MoveL 1052 to (0, 54.97, 50) mm, rotated rx 180 ry 0 rz 180 deg; joints [-152.438, -60.713, -86.238, 31.91, 61.088, -16.755]
  Call Extruder(10810.73949)
  MoveL 1053 to (-12.23, 53.59, 50) mm, rotated rx 180 ry 0 rz 180 deg; joints [-151.764, -60.094, -88.252, 32.246, 62.462, -16.26]
  Call Extruder(10821.66963)
  MoveL 1054 to (-23.85, 49.52, 50) mm, rotated rx 180 ry 0 rz 180 deg; joints [-151.463, -59.479, -90.349, 32.17, 63.798, -15.521]
  Call Extruder(10832.59991)
  MoveL 1055 to (-34.27, 42.98, 50) mm, rotated rx 180 ry 0 rz 180 deg; joints [-151.589, -58.902, -92.428, 31.655, 65.04, -14.583]
  Call Extruder(10843.53003)
  MoveL 1056 to (-42.98, 34.27, 50) mm, rotated rx -180 ry 0 rz -180 deg; joints [-152.179, -58.391, -94.383, 30.687, 66.133, -13.502]
  Call Extruder(10854.46031)
  MoveL 1057 to (-49.53, 23.85, 50) mm, rotated rx -180 ry 0 rz 180 deg; joints [-153.248, -57.967, -96.114, 29.27, 67.025, -12.34]
  Call Extruder(10865.39045)
  MoveL 1058 to (-53.59, 12.23, 50) mm, rotated rx 180 ry 0 rz 180 deg; joints [-154.769, -57.643, -97.52, 27.44, 67.669, -11.161]
  Call Extruder(10876.32067)
  MoveL 1059 to (-54.97, 0, 50) mm, rotated rx -180 ry 0 rz -180 deg; joints [-156.673, -57.426, -98.52, 25.279, 68.02, -10.024]
  Call Extruder(10881.84629)
  MoveL 1060 to (-54.27, -6.18, 50) mm, rotated rx 180 ry 0 rz 180 deg; joints [-157.76, -57.367, -98.797, 24.086, 68.035, -9.493]
  Set speed (130.0 mm/s)
  MoveL 1061 to (-49.9, -9.51, 50) mm, rotated rx 180 ry 0 rz -180 deg; joints [-158.616, -57.462, -98.351, 23.231, 67.572, -9.301]
  MoveL 1062 to (2.97, -12.99, 50) mm, rotated rx 180 ry 0 rz -180 deg; joints [-162.152, -59.481, -90.344, 20.428, 61.416, -10.104]
  Call Extruder(10886.50986)
  Set speed (80.0 mm/s)
  MoveL 1063 to (5.78, -12.01, 50) mm, rotated rx -180 ry 0 rz 180 deg; joints [-162.141, -59.628, -89.833, 20.511, 61.077, -10.256]
  Call Extruder(10891.17348)
  MoveL 1064 to (8.31, -10.42, 50) mm, rotated rx 180 ry 0 rz -180 deg; joints [-162.027, -59.773, -89.336, 20.708, 60.767, -10.46]
  Call Extruder(10895.83767)
  MoveL 1065 to (10.42, -8.31, 50) mm, rotated rx -180 ry 0 rz 180 deg; joints [-161.819, -59.908, -88.876, 21.008, 60.502, -10.707]
  Call Extruder(10900.50130)
  MoveL 1066 to (12.01, -5.78, 50) mm, rotated rx 180 ry 0 rz 180 deg; joints [-161.529, -60.027, -88.476, 21.393, 60.295, -10.986]
  Call Extruder(10905.16487)
  MoveL 1067 to (12.99, -2.97, 50) mm, rotated rx -180 ry 0 rz -180 deg; joints [-161.171, -60.123, -88.157, 21.845, 60.156, -11.282]
  Call Extruder(10909.82882)
  MoveL 1068 to (13.33, 0, 50) mm, rotated rx -180 ry 0 rz 180 deg; joints [-160.763, -60.19, -87.933, 22.34, 60.092, -11.58]
  Call Extruder(10914.49277)
  MoveL 1069 to (13, 2.97, 50) mm, rotated rx 180 ry 0 rz -180 deg; joints [-160.324, -60.226, -87.815, 22.854, 60.106, -11.863]
  Call Extruder(10919.15635)
  MoveL 1070 to (12.01, 5.78, 50) mm, rotated rx 180 ry 0 rz -180 deg; joints [-159.874, -60.228, -87.81, 23.362, 60.195, -12.118]
  Call Extruder(10923.81997)
  MoveL 1071 to (10.42, 8.31, 50) mm, rotated rx 180 ry 0 rz 180 deg; joints [-159.432, -60.195, -87.916, 23.842, 60.357, -12.329]
  Call Extruder(10928.48416)
  MoveL 1072 to (8.31, 10.42, 50) mm, rotated rx 180 ry 0 rz 180 deg; joints [-159.021, -60.131, -88.13, 24.27, 60.582, -12.487]
  Call Extruder(10933.14778)
  MoveL 1073 to (5.78, 12.01, 50) mm, rotated rx 180 ry 0 rz 180 deg; joints [-158.657, -60.038, -88.441, 24.626, 60.859, -12.583]
  Call Extruder(10937.81136)
  MoveL 1074 to (2.97, 12.99, 50) mm, rotated rx 180 ry 0 rz 180 deg; joints [-158.359, -59.921, -88.833, 24.894, 61.174, -12.612]
  Call Extruder(10942.47532)
  MoveL 1075 to (0, 13.33, 50) mm, rotated rx -180 ry 0 rz 180 deg; joints [-158.143, -59.787, -89.288, 25.061, 61.512, -12.574]
  Call Extruder(10947.13927)
  MoveL 1076 to (-2.97, 12.99, 50) mm, rotated rx 180 ry 0 rz 180 deg; joints [-158.019, -59.642, -89.783, 25.118, 61.856, -12.47]
  Call Extruder(10951.80283)
  MoveL 1077 to (-5.78, 12.01, 50) mm, rotated rx 180 ry 0 rz 180 deg; joints [-157.997, -59.495, -90.294, 25.06, 62.19, -12.306]
  Call Extruder(10956.46646)
  MoveL 1078 to (-8.31, 10.42, 50) mm, rotated rx 180 ry 0 rz 180 deg; joints [-158.08, -59.353, -90.795, 24.89, 62.498, -12.093]
  Call Extruder(10961.13066)
  MoveL 1079 to (-10.42, 8.31, 50) mm, rotated rx 180 ry 0 rz 180 deg; joints [-158.266, -59.222, -91.261, 24.612, 62.763, -11.841]
  Call Extruder(10965.79428)
  MoveL 1080 to (-12.01, 5.78, 50) mm, rotated rx 180 ry 0 rz -180 deg; joints [-158.549, -59.109, -91.668, 24.239, 62.974, -11.562]
  Call Extruder(10970.45785)
  MoveL 1081 to (-13, 2.97, 50) mm, rotated rx 180 ry 0 rz -180 deg; joints [-158.913, -59.019, -91.995, 23.789, 63.119, -11.272]
  Call Extruder(10975.12181)
  MoveL 1082 to (-13.33, 0, 50) mm, rotated rx 180 ry 0 rz 180 deg; joints [-159.341, -58.957, -92.225, 23.284, 63.189, -10.985]
  Call Extruder(10979.78576)
  MoveL 1083 to (-12.99, -2.97, 50) mm, rotated rx 180 ry 0 rz 180 deg; joints [-159.811, -58.924, -92.346, 22.75, 63.183, -10.713]
  Call Extruder(10984.44933)
  MoveL 1084 to (-12.01, -5.78, 50) mm, rotated rx 180 ry 0 rz 180 deg; joints [-160.294, -58.922, -92.352, 22.216, 63.097, -10.47]
  Call Extruder(10989.11295)
  MoveL 1085 to (-10.42, -8.31, 50) mm, rotated rx 180 ry 0 rz 180 deg; joints [-160.766, -58.952, -92.242, 21.711, 62.938, -10.268]
  Call Extruder(10993.77714)
  MoveL 1086 to (-8.31, -10.42, 50) mm, rotated rx 180 ry 0 rz -180 deg; joints [-161.2, -59.012, -92.022, 21.261, 62.713, -10.114]
  Call Extruder(10998.44078)
  MoveL 1087 to (-5.78, -12.01, 50) mm, rotated rx 180 ry 0 rz 180 deg; joints [-161.572, -59.099, -91.704, 20.892, 62.432, -10.018]
  Call Extruder(11003.10435)
  MoveL 1088 to (-2.97, -12.99, 50) mm, rotated rx 180 ry 0 rz 180 deg; joints [-161.863, -59.21, -91.304, 20.622, 62.111, -9.983]
  Call Extruder(11007.76828)
  MoveL 1089 to (0, -13.33, 50) mm, rotated rx -180 ry 0 rz -180 deg; joints [-162.059, -59.339, -90.843, 20.465, 61.767, -10.012]
  Call Extruder(11012.43225)
  MoveL 1090 to (2.97, -12.99, 50) mm, rotated rx 180 ry 0 rz -180 deg; joints [-162.152, -59.481, -90.344, 20.428, 61.416, -10.104]
  Set speed (130.0 mm/s)
  MoveL 1091 to (2.97, -12.99, 55) mm, rotated rx 180 ry 0 rz -180 deg; joints [-162.152, -58.714, -90.747, 20.498, 61.075, -10.249]
  MoveL 1092 to (-26.25, -4.54, 55) mm, rotated rx 180 ry 0 rz 180 deg; joints [-159.288, -57.567, -94.911, 23.091, 64.391, -10.441]
  Call Extruder(11014.66488)
  Set speed (60.0 mm/s)
  MoveL 1093 to (-26.09, -5.96, 55) mm, rotated rx 180 ry 0 rz 180 deg; joints [-159.522, -57.552, -94.968, 22.829, 64.388, -10.313]
  Call Extruder(11024.02967)
  MoveL 1094 to (-24.11, -11.61, 55) mm, rotated rx 180 ry 0 rz -180 deg; joints [-160.532, -57.549, -94.98, 21.723, 64.22, -9.831]
  Call Extruder(11033.39459)
  MoveL 1095 to (-20.93, -16.69, 55) mm, rotated rx 180 ry 0 rz 180 deg; joints [-161.513, -57.607, -94.755, 20.677, 63.9, -9.427]
  Call Extruder(11042.75979)
  MoveL 1096 to (-16.69, -20.93, 55) mm, rotated rx -180 ry 0 rz -180 deg; joints [-162.406, -57.725, -94.306, 19.75, 63.445, -9.119]
  Call Extruder(11052.12472)
  MoveL 1097 to (-11.61, -24.12, 55) mm, rotated rx 180 ry 0 rz 180 deg; joints [-163.159, -57.897, -93.657, 18.996, 62.878, -8.919]
  Call Extruder(11061.48950)
  MoveL 1098 to (-5.96, -26.09, 55) mm, rotated rx 180 ry 0 rz 180 deg; joints [-163.733, -58.119, -92.845, 18.456, 62.229, -8.839]
  Call Extruder(11070.85461)
  MoveL 1099 to (0, -26.77, 55) mm, rotated rx 180 ry 0 rz 180 deg; joints [-164.103, -58.379, -91.911, 18.154, 61.533, -8.883]
  Call Extruder(11071.92859)
  MoveL 1100 to (0.68, -26.69, 55) mm, rotated rx 180 ry 0 rz 180 deg; joints [-164.121, -58.412, -91.796, 18.148, 61.452, -8.903]
  Call Extruder(11080.21972)
  MoveL 1101 to (5.96, -26.09, 55) mm, rotated rx -180 ry 0 rz 180 deg; joints [-164.258, -58.668, -90.905, 18.103, 60.827, -9.054]
  Call Extruder(11089.58452)
  MoveL 1102 to (11.61, -24.12, 55) mm, rotated rx 180 ry 0 rz 180 deg; joints [-164.201, -58.969, -89.878, 18.296, 60.147, -9.346]
  Call Extruder(11098.94943)
  MoveL 1103 to (16.69, -20.93, 55) mm, rotated rx 180 ry 0 rz 180 deg; joints [-163.944, -59.27, -88.881, 18.718, 59.529, -9.749]
  Call Extruder(11108.31463)
  MoveL 1104 to (20.93, -16.69, 55) mm, rotated rx 180 ry 0 rz 180 deg; joints [-163.508, -59.552, -87.962, 19.34, 59.003, -10.246]
  Call Extruder(11117.67956)
  MoveL 1105 to (24.12, -11.61, 55) mm, rotated rx 180 ry 0 rz 180 deg; joints [-162.92, -59.801, -87.166, 20.128, 58.595, -10.812]
  Call Extruder(11127.04435)
  MoveL 1106 to (26.09, -5.96, 55) mm, rotated rx 180 ry 0 rz -180 deg; joints [-162.209, -60.003, -86.53, 21.04, 58.326, -11.419]
  Call Extruder(11136.40945)
  MoveL 1107 to (26.77, 0, 55) mm, rotated rx 180 ry 0 rz -180 deg; joints [-161.41, -60.146, -86.085, 22.028, 58.207, -12.033]
  Call Extruder(11145.77456)
  MoveL 1108 to (26.09, 5.96, 55) mm, rotated rx 180 ry 0 rz 180 deg; joints [-160.556, -60.221, -85.851, 23.047, 58.243, -12.621]
  Call Extruder(11155.13936)
  MoveL 1109 to (24.11, 11.61, 55) mm, rotated rx 180 ry 0 rz 180 deg; joints [-159.683, -60.225, -85.84, 24.049, 58.431, -13.15]
  Call Extruder(11164.50427)
  MoveL 1110 to (20.93, 16.69, 55) mm, rotated rx 180 ry 0 rz 180 deg; joints [-158.826, -60.156, -86.052, 24.99, 58.76, -13.59]
  Call Extruder(11173.86948)
  MoveL 1111 to (16.69, 20.93, 55) mm, rotated rx 180 ry 0 rz 180 deg; joints [-158.019, -60.02, -86.477, 25.83, 59.212, -13.916]
  Call Extruder(11183.23439)
  MoveL 1112 to (11.61, 24.11, 55) mm, rotated rx 180 ry 0 rz 180 deg; joints [-157.299, -59.824, -87.095, 26.531, 59.765, -14.112]
  Call Extruder(11192.59919)
  MoveL 1113 to (5.96, 26.09, 55) mm, rotated rx -180 ry 0 rz -180 deg; joints [-156.697, -59.579, -87.877, 27.065, 60.391, -14.168]
  Call Extruder(11201.96430)
  MoveL 1114 to (0, 26.77, 55) mm, rotated rx -180 ry 0 rz 180 deg; joints [-156.245, -59.299, -88.785, 27.407, 61.061, -14.084]
  Call Extruder(11211.32940)
  MoveL 1115 to (-5.96, 26.09, 55) mm, rotated rx 180 ry 0 rz 180 deg; joints [-155.969, -59, -89.777, 27.537, 61.742, -13.866]
  Call Extruder(11220.69419)
  MoveL 1116 to (-11.61, 24.12, 55) mm, rotated rx -180 ry 0 rz -180 deg; joints [-155.891, -58.697, -90.803, 27.446, 62.402, -13.528]
  Call Extruder(11230.05911)
  MoveL 1117 to (-16.69, 20.93, 55) mm, rotated rx 180 ry 0 rz -180 deg; joints [-156.025, -58.407, -91.814, 27.129, 63.012, -13.09]
  Call Extruder(11239.42432)
  MoveL 1118 to (-20.93, 16.69, 55) mm, rotated rx -180 ry 0 rz 180 deg; joints [-156.374, -58.143, -92.757, 26.594, 63.54, -12.575]
  Call Extruder(11248.78923)
  MoveL 1119 to (-24.11, 11.61, 55) mm, rotated rx -180 ry 0 rz 180 deg; joints [-156.928, -57.917, -93.583, 25.859, 63.961, -12.012]
  Call Extruder(11258.15403)
  MoveL 1120 to (-26.09, 5.96, 55) mm, rotated rx 180 ry 0 rz 180 deg; joints [-157.665, -57.74, -94.25, 24.955, 64.253, -11.428]
  Call Extruder(11267.51914)
  MoveL 1121 to (-26.77, 0, 55) mm, rotated rx 180 ry 0 rz 180 deg; joints [-158.546, -57.616, -94.72, 23.927, 64.399, -10.853]
  Call Extruder(11272.30787)
  MoveL 1122 to (-26.42, -3.05, 55) mm, rotated rx -180 ry 0 rz 180 deg; joints [-159.044, -57.583, -94.849, 23.366, 64.393, -10.577]
  Set speed (130.0 mm/s)
  MoveL 1123 to (-41.86, -6.3, 55) mm, rotated rx -180 ry 0 rz 180 deg; joints [-158.606, -56.955, -97.386, 23.492, 66.224, -9.939]
  Call Extruder(11277.30572)
  Set speed (60.0 mm/s)
  MoveL 1124 to (-41.51, -9.47, 55) mm, rotated rx -180 ry 0 rz -180 deg; joints [-159.151, -56.924, -97.517, 22.887, 66.222, -9.659]
  Call Extruder(11292.20137)
  MoveL 1125 to (-38.36, -18.47, 55) mm, rotated rx 180 ry 0 rz 180 deg; joints [-160.835, -56.92, -97.536, 21.066, 65.964, -8.917]
  Call Extruder(11307.09723)
  MoveL 1126 to (-33.29, -26.54, 55) mm, rotated rx -180 ry 0 rz 180 deg; joints [-162.466, -57.006, -97.17, 19.342, 65.458, -8.295]
  Call Extruder(11321.99304)
  MoveL 1127 to (-26.54, -33.28, 55) mm, rotated rx 180 ry 0 rz -180 deg; joints [-163.93, -57.182, -96.441, 17.825, 64.728, -7.816]
  Call Extruder(11336.88890)
  MoveL 1128 to (-18.47, -38.36, 55) mm, rotated rx -180 ry 0 rz 180 deg; joints [-165.137, -57.444, -95.392, 16.61, 63.815, -7.499]
  Call Extruder(11351.78454)
  MoveL 1129 to (-9.47, -41.5, 55) mm, rotated rx 180 ry 0 rz -180 deg; joints [-166.024, -57.784, -94.083, 15.76, 62.77, -7.358]
  Call Extruder(11366.68042)
  MoveL 1130 to (0, -42.57, 55) mm, rotated rx 180 ry 0 rz 180 deg; joints [-166.562, -58.19, -92.587, 15.311, 61.651, -7.407]
  Call Extruder(11370.51995)
  MoveL 1131 to (2.44, -42.3, 55) mm, rotated rx 180 ry 0 rz 180 deg; joints [-166.61, -58.305, -92.176, 15.299, 61.359, -7.47]
  Call Extruder(11381.57629)
  MoveL 1132 to (9.47, -41.51, 55) mm, rotated rx -180 ry 0 rz 180 deg; joints [-166.745, -58.645, -90.983, 15.271, 60.518, -7.653]
  Call Extruder(11396.47195)
  MoveL 1133 to (18.47, -38.36, 55) mm, rotated rx 180 ry 0 rz 180 deg; joints [-166.591, -59.127, -89.351, 15.624, 59.432, -8.095]
  Call Extruder(11411.36780)
  MoveL 1134 to (26.54, -33.29, 55) mm, rotated rx 180 ry 0 rz 180 deg; joints [-166.133, -59.611, -87.773, 16.335, 58.446, -8.72]
  Call Extruder(11426.26362)
  MoveL 1135 to (33.28, -26.54, 55) mm, rotated rx 180 ry 0 rz 180 deg; joints [-165.409, -60.069, -86.323, 17.357, 57.611, -9.504]
  Call Extruder(11441.15947)
  MoveL 1136 to (38.36, -18.47, 55) mm, rotated rx 180 ry 0 rz 180 deg; joints [-164.468, -60.476, -85.068, 18.627, 56.968, -10.411]
  Call Extruder(11456.05512)
  MoveL 1137 to (41.51, -9.47, 55) mm, rotated rx 180 ry 0 rz 180 deg; joints [-163.355, -60.807, -84.068, 20.079, 56.547, -11.393]
  Call Extruder(11470.95099)
  MoveL 1138 to (42.57, 0, 55) mm, rotated rx 180 ry 0 rz 180 deg; joints [-162.12, -61.042, -83.368, 21.639, 56.367, -12.393]
  Call Extruder(11485.84687)
  MoveL 1139 to (41.5, 9.47, 55) mm, rotated rx 180 ry 0 rz 180 deg; joints [-160.81, -61.166, -83.001, 23.233, 56.434, -13.352]
  Call Extruder(11500.74253)
  MoveL 1140 to (38.36, 18.47, 55) mm, rotated rx -180 ry 0 rz 180 deg; joints [-159.475, -61.172, -82.983, 24.791, 56.741, -14.214]
  Call Extruder(11515.63837)
  MoveL 1141 to (33.29, 26.54, 55) mm, rotated rx 180 ry 0 rz 180 deg; joints [-158.16, -61.059, -83.316, 26.245, 57.271, -14.926]
  Call Extruder(11530.53420)
  MoveL 1142 to (26.54, 33.28, 55) mm, rotated rx -180 ry 0 rz 180 deg; joints [-156.916, -60.835, -83.984, 27.54, 57.993, -15.45]
  Call Extruder(11545.43004)
  MoveL 1143 to (18.47, 38.36, 55) mm, rotated rx -180 ry 0 rz -180 deg; joints [-155.789, -60.513, -84.957, 28.626, 58.87, -15.758]
  Call Extruder(11560.32570)
  MoveL 1144 to (9.47, 41.51, 55) mm, rotated rx -180 ry 0 rz 180 deg; joints [-154.828, -60.112, -86.188, 29.462, 59.858, -15.836]
  Call Extruder(11575.22158)
  MoveL 1145 to (0, 42.57, 55) mm, rotated rx 180 ry 0 rz 180 deg; joints [-154.081, -59.658, -87.622, 30.013, 60.911, -15.686]
  Call Extruder(11590.11745)
  MoveL 1146 to (-9.47, 41.51, 55) mm, rotated rx 180 ry 0 rz -180 deg; joints [-153.594, -59.176, -89.191, 30.25, 61.981, -15.321]
  Call Extruder(11605.01310)
  MoveL 1147 to (-18.47, 38.36, 55) mm, rotated rx 180 ry 0 rz 180 deg; joints [-153.408, -58.692, -90.821, 30.152, 63.02, -14.764]
  Call Extruder(11619.90896)
  MoveL 1148 to (-26.54, 33.29, 55) mm, rotated rx -180 ry 0 rz 180 deg; joints [-153.557, -58.233, -92.431, 29.704, 63.981, -14.05]
  Call Extruder(11634.80477)
  MoveL 1149 to (-33.28, 26.54, 55) mm, rotated rx 180 ry 0 rz -180 deg; joints [-154.059, -57.821, -93.941, 28.906, 64.821, -13.22]
  Call Extruder(11649.70062)
  MoveL 1150 to (-38.36, 18.47, 55) mm, rotated rx -180 ry 0 rz 180 deg; joints [-154.913, -57.474, -95.272, 27.772, 65.497, -12.32]
  Call Extruder(11664.59628)
  MoveL 1151 to (-41.5, 9.47, 55) mm, rotated rx 180 ry 0 rz 180 deg; joints [-156.091, -57.204, -96.35, 26.342, 65.975, -11.398]
  Call Extruder(11679.49215)
  MoveL 1152 to (-42.57, 0, 55) mm, rotated rx 180 ry 0 rz -180 deg; joints [-157.533, -57.02, -97.113, 24.683, 66.224, -10.497]
  Call Extruder(11687.04643)
  MoveL 1153 to (-42.03, -4.8, 55) mm, rotated rx 180 ry 0 rz 180 deg; joints [-158.35, -56.97, -97.324, 23.775, 66.224, -10.071]
  Set speed (130.0 mm/s)
  MoveL 1154 to (-54.1, -7.67, 55) mm, rotated rx 180 ry 0 rz 180 deg; joints [-158.024, -56.526, -99.284, 23.864, 67.667, -9.542]
  Call Extruder(11691.11906)
  Set speed (30.0 mm/s)
  MoveL 1155 to (-53.59, -12.23, 55) mm, rotated rx 180 ry 0 rz 180 deg; joints [-158.835, -56.486, -99.473, 22.974, 67.672, -9.15]
  Call Extruder(11702.04919)
  MoveL 1156 to (-49.52, -23.85, 55) mm, rotated rx 180 ry 0 rz 180 deg; joints [-161.095, -56.48, -99.498, 20.553, 67.349, -8.217]
  Call Extruder(11712.97948)
  MoveL 1157 to (-42.98, -34.27, 55) mm, rotated rx 180 ry 0 rz 180 deg; joints [-163.275, -56.585, -99.016, 18.261, 66.696, -7.437]
  Call Extruder(11723.90960)
  MoveL 1158 to (-34.27, -42.98, 55) mm, rotated rx 180 ry 0 rz 180 deg; joints [-165.21, -56.799, -98.058, 16.26, 65.745, -6.832]
  Call Extruder(11734.83988)
  MoveL 1159 to (-23.85, -49.53, 55) mm, rotated rx 180 ry 0 rz 180 deg; joints [-166.774, -57.123, -96.684, 14.678, 64.552, -6.421]
  Call Extruder(11745.77001)
  MoveL 1160 to (-12.23, -53.59, 55) mm, rotated rx 180 ry 0 rz 180 deg; joints [-167.889, -57.55, -94.978, 13.597, 63.189, -6.226]
  Call Extruder(11756.70024)
  MoveL 1161 to (0, -54.97, 55) mm, rotated rx 180 ry 0 rz 180 deg; joints [-168.526, -58.066, -93.036, 13.053, 61.732, -6.266]
  Call Extruder(11760.11472)
  MoveL 1162 to (3.82, -54.54, 55) mm, rotated rx -180 ry 0 rz 180 deg; joints [-168.581, -58.244, -92.392, 13.048, 61.272, -6.356]
  Call Extruder(11767.63046)
  MoveL 1163 to (12.23, -53.59, 55) mm, rotated rx -180 ry 0 rz 180 deg; joints [-168.697, -58.651, -90.961, 13.046, 60.262, -6.557]
  Call Extruder(11778.56060)
  MoveL 1164 to (23.85, -49.53, 55) mm, rotated rx 180 ry 0 rz 180 deg; joints [-168.436, -59.276, -88.859, 13.545, 58.855, -7.103]
  Call Extruder(11789.49088)
  MoveL 1165 to (34.27, -42.98, 55) mm, rotated rx 180 ry 0 rz 180 deg; joints [-167.797, -59.908, -86.829, 14.501, 57.582, -7.894]
  Call Extruder(11800.42100)
  MoveL 1166 to (42.98, -34.27, 55) mm, rotated rx 180 ry 0 rz 180 deg; joints [-166.837, -60.509, -84.967, 15.847, 56.506, -8.903]
  Call Extruder(11811.35128)
  MoveL 1167 to (49.53, -23.85, 55) mm, rotated rx -180 ry 0 rz 180 deg; joints [-165.618, -61.045, -83.359, 17.502, 55.679, -10.082]
  Call Extruder(11822.28142)
  MoveL 1168 to (53.59, -12.23, 55) mm, rotated rx -180 ry 0 rz -180 deg; joints [-164.2, -61.481, -82.077, 19.379, 55.141, -11.368]
  Call Extruder(11833.21164)
  MoveL 1169 to (54.97, 0, 55) mm, rotated rx -180 ry 0 rz 180 deg; joints [-162.641, -61.792, -81.18, 21.384, 54.916, -12.684]
  Call Extruder(11844.14186)
  MoveL 1170 to (53.59, 12.23, 55) mm, rotated rx 180 ry 0 rz 180 deg; joints [-160.996, -61.956, -80.709, 23.42, 55.012, -13.948]
  Call Extruder(11855.07200)
  MoveL 1171 to (49.52, 23.85, 55) mm, rotated rx 180 ry 0 rz -180 deg; joints [-159.322, -61.964, -80.687, 25.397, 55.418, -15.082]
  Call Extruder(11866.00228)
  MoveL 1172 to (42.98, 34.27, 55) mm, rotated rx -180 ry 0 rz 180 deg; joints [-157.673, -61.815, -81.114, 27.236, 56.109, -16.014]
  Call Extruder(11876.93240)
  MoveL 1173 to (34.27, 42.98, 55) mm, rotated rx 180 ry 0 rz 180 deg; joints [-156.102, -61.518, -81.97, 28.868, 57.045, -16.694]
  Call Extruder(11887.86268)
  MoveL 1174 to (23.85, 49.52, 55) mm, rotated rx -180 ry 0 rz 180 deg; joints [-154.667, -61.093, -83.216, 30.237, 58.176, -17.085]
  Call Extruder(11898.79282)
  MoveL 1175 to (12.23, 53.59, 55) mm, rotated rx 180 ry 0 rz 180 deg; joints [-153.426, -60.566, -84.795, 31.298, 59.445, -17.174]
  Call Extruder(11909.72304)
  MoveL 1176 to (0, 54.97, 55) mm, rotated rx -180 ry 0 rz 180 deg; joints [-152.438, -59.969, -86.635, 32.012, 60.794, -16.964]
  Call Extruder(11920.65327)
  MoveL 1177 to (-12.23, 53.59, 55) mm, rotated rx 180 ry 0 rz 180 deg; joints [-151.764, -59.339, -88.652, 32.345, 62.162, -16.474]
  Call Extruder(11931.58340)
  MoveL 1178 to (-23.85, 49.52, 55) mm, rotated rx 180 ry 0 rz 180 deg; joints [-151.463, -58.712, -90.752, 32.266, 63.49, -15.738]
  Call Extruder(11942.51368)
  MoveL 1179 to (-34.27, 42.98, 55) mm, rotated rx -180 ry 0 rz 180 deg; joints [-151.589, -58.122, -92.834, 31.747, 64.722, -14.8]
  Call Extruder(11953.44380)
  MoveL 1180 to (-42.98, 34.27, 55) mm, rotated rx -180 ry 0 rz -180 deg; joints [-152.179, -57.597, -94.794, 30.774, 65.804, -13.716]
  Call Extruder(11964.37408)
  MoveL 1181 to (-49.53, 23.85, 55) mm, rotated rx 180 ry 0 rz -180 deg; joints [-153.248, -57.161, -96.528, 29.351, 66.684, -12.548]
  Call Extruder(11975.30422)
  MoveL 1182 to (-53.59, 12.23, 55) mm, rotated rx 180 ry 0 rz -180 deg; joints [-154.769, -56.826, -97.939, 27.516, 67.316, -11.36]
  Call Extruder(11986.23444)
  MoveL 1183 to (-54.97, 0, 55) mm, rotated rx -180 ry 0 rz -180 deg; joints [-156.673, -56.601, -98.942, 25.349, 67.655, -10.21]
  Call Extruder(11991.76006)
  MoveL 1184 to (-54.27, -6.18, 55) mm, rotated rx 180 ry 0 rz -180 deg; joints [-157.76, -56.54, -99.22, 24.154, 67.665, -9.671]
  Set speed (130.0 mm/s)
  MoveL 1185 to (-49.9, -9.51, 55) mm, rotated rx -180 ry 0 rz -180 deg; joints [-158.616, -56.638, -98.771, 23.298, 67.202, -9.473]
  MoveL 1186 to (2.97, -12.99, 55) mm, rotated rx 180 ry 0 rz -180 deg; joints [-162.152, -58.714, -90.747, 20.498, 61.075, -10.249]
  Call Extruder(11996.42363)
  Set speed (80.0 mm/s)
  MoveL 1187 to (5.78, -12.01, 55) mm, rotated rx 180 ry 0 rz 180 deg; joints [-162.141, -58.864, -90.236, 20.582, 60.738, -10.401]
  Call Extruder(12001.08725)
  MoveL 1188 to (8.31, -10.42, 55) mm, rotated rx 180 ry 0 rz -180 deg; joints [-162.027, -59.012, -89.737, 20.78, 60.431, -10.606]
  Call Extruder(12005.75144)
  MoveL 1189 to (10.42, -8.31, 55) mm, rotated rx 180 ry 0 rz 180 deg; joints [-161.819, -59.15, -89.276, 21.081, 60.168, -10.855]
  Call Extruder(12010.41507)
  MoveL 1190 to (12.01, -5.78, 55) mm, rotated rx 180 ry 0 rz -180 deg; joints [-161.529, -59.271, -88.876, 21.468, 59.964, -11.136]
  Call Extruder(12015.07864)
  MoveL 1191 to (13, -2.97, 55) mm, rotated rx -180 ry 0 rz -180 deg; joints [-161.171, -59.369, -88.556, 21.921, 59.827, -11.434]
  Call Extruder(12019.74259)
  MoveL 1192 to (13.33, 0, 55) mm, rotated rx -180 ry 0 rz 180 deg; joints [-160.763, -59.438, -88.332, 22.418, 59.765, -11.735]
  Call Extruder(12024.40655)
  MoveL 1193 to (12.99, 2.97, 55) mm, rotated rx -180 ry 0 rz 180 deg; joints [-160.324, -59.474, -88.214, 22.933, 59.781, -12.022]
  Call Extruder(12029.07012)
  MoveL 1194 to (12.01, 5.78, 55) mm, rotated rx 180 ry 0 rz -180 deg; joints [-159.874, -59.476, -88.209, 23.443, 59.872, -12.279]
  Call Extruder(12033.73374)
  MoveL 1195 to (10.42, 8.31, 55) mm, rotated rx 180 ry 0 rz 180 deg; joints [-159.432, -59.443, -88.316, 23.924, 60.034, -12.494]
  Call Extruder(12038.39794)
  MoveL 1196 to (8.31, 10.42, 55) mm, rotated rx 180 ry 0 rz 180 deg; joints [-159.021, -59.377, -88.53, 24.352, 60.259, -12.655]
  Call Extruder(12043.06156)
  MoveL 1197 to (5.78, 12.01, 55) mm, rotated rx 180 ry 0 rz -180 deg; joints [-158.657, -59.282, -88.841, 24.709, 60.536, -12.753]
  Call Extruder(12047.72513)
  MoveL 1198 to (2.97, 12.99, 55) mm, rotated rx -180 ry 0 rz 180 deg; joints [-158.359, -59.163, -89.234, 24.978, 60.85, -12.785]
  Call Extruder(12052.38909)
  MoveL 1199 to (0, 13.33, 55) mm, rotated rx -180 ry 0 rz -180 deg; joints [-158.143, -59.026, -89.689, 25.145, 61.186, -12.747]
  Call Extruder(12057.05304)
  MoveL 1200 to (-2.97, 13, 55) mm, rotated rx 180 ry 0 rz -180 deg; joints [-158.019, -58.878, -90.185, 25.201, 61.529, -12.644]
  Call Extruder(12061.71661)
  MoveL 1201 to (-5.78, 12.01, 55) mm, rotated rx -180 ry 0 rz 180 deg; joints [-157.997, -58.728, -90.697, 25.142, 61.861, -12.481]
  Call Extruder(12066.38024)
  MoveL 1202 to (-8.31, 10.42, 55) mm, rotated rx -180 ry 0 rz 180 deg; joints [-158.08, -58.583, -91.199, 24.97, 62.166, -12.267]
  Call Extruder(12071.04443)
  MoveL 1203 to (-10.42, 8.31, 55) mm, rotated rx -180 ry 0 rz 180 deg; joints [-158.266, -58.449, -91.665, 24.691, 62.429, -12.014]
  Call Extruder(12075.70805)
  MoveL 1204 to (-12.01, 5.78, 55) mm, rotated rx 180 ry 0 rz 180 deg; joints [-158.549, -58.334, -92.073, 24.317, 62.637, -11.733]
  Call Extruder(12080.37162)
  MoveL 1205 to (-12.99, 2.97, 55) mm, rotated rx 180 ry 0 rz -180 deg; joints [-158.913, -58.242, -92.401, 23.866, 62.779, -11.441]
  Call Extruder(12085.03558)
  MoveL 1206 to (-13.33, 0, 55) mm, rotated rx 180 ry 0 rz -180 deg; joints [-159.341, -58.178, -92.631, 23.359, 62.847, -11.15]
  Call Extruder(12089.69953)
  MoveL 1207 to (-12.99, -2.97, 55) mm, rotated rx 180 ry 0 rz 180 deg; joints [-159.811, -58.144, -92.752, 22.824, 62.838, -10.875]
  Call Extruder(12094.36310)
  MoveL 1208 to (-12.01, -5.78, 55) mm, rotated rx -180 ry 0 rz 180 deg; joints [-160.294, -58.143, -92.758, 22.289, 62.752, -10.629]
  Call Extruder(12099.02673)
  MoveL 1209 to (-10.42, -8.31, 55) mm, rotated rx -180 ry 0 rz 180 deg; joints [-160.766, -58.173, -92.648, 21.782, 62.592, -10.423]
  Call Extruder(12103.69092)
  MoveL 1210 to (-8.31, -10.42, 55) mm, rotated rx 180 ry 0 rz 180 deg; joints [-161.2, -58.234, -92.428, 21.332, 62.366, -10.267]
  Call Extruder(12108.35455)
  MoveL 1211 to (-5.78, -12.01, 55) mm, rotated rx -180 ry 0 rz 180 deg; joints [-161.572, -58.324, -92.109, 20.962, 62.086, -10.167]
  Call Extruder(12113.01811)
  MoveL 1212 to (-2.97, -12.99, 55) mm, rotated rx -180 ry 0 rz 180 deg; joints [-161.863, -58.437, -91.709, 20.691, 61.767, -10.13]
  Call Extruder(12117.68206)
  MoveL 1213 to (0, -13.33, 55) mm, rotated rx 180 ry 0 rz -180 deg; joints [-162.059, -58.569, -91.247, 20.535, 61.423, -10.158]
  Call Extruder(12122.34603)
  MoveL 1214 to (2.97, -12.99, 55) mm, rotated rx 180 ry 0 rz -180 deg; joints [-162.152, -58.714, -90.747, 20.498, 61.075, -10.249]
  Set speed (130.0 mm/s)
  MoveL 1215 to (2.97, -12.99, 60) mm, rotated rx 180 ry 0 rz -180 deg; joints [-162.152, -57.947, -91.141, 20.571, 60.725, -10.399]
  MoveL 1216 to (-26.25, -4.54, 60) mm, rotated rx 180 ry 0 rz 180 deg; joints [-159.288, -56.772, -95.313, 23.166, 64.029, -10.613]
  Call Extruder(12124.57865)
  Set speed (60.0 mm/s)
  MoveL 1217 to (-26.09, -5.96, 60) mm, rotated rx 180 ry 0 rz 180 deg; joints [-159.522, -56.757, -95.37, 22.902, 64.026, -10.483]
  Call Extruder(12133.94344)
  MoveL 1218 to (-24.11, -11.61, 60) mm, rotated rx -180 ry 0 rz 180 deg; joints [-160.532, -56.754, -95.382, 21.794, 63.854, -9.993]
  Call Extruder(12143.30836)
  MoveL 1219 to (-20.93, -16.69, 60) mm, rotated rx 180 ry 0 rz 180 deg; joints [-161.513, -56.813, -95.157, 20.745, 63.533, -9.582]
  Call Extruder(12152.67356)
  MoveL 1220 to (-16.69, -20.93, 60) mm, rotated rx -180 ry 0 rz -180 deg; joints [-162.406, -56.934, -94.707, 19.816, 63.078, -9.267]
  Call Extruder(12162.03849)
  MoveL 1221 to (-11.61, -24.12, 60) mm, rotated rx -180 ry 0 rz 180 deg; joints [-163.159, -57.111, -94.057, 19.061, 62.512, -9.061]
  Call Extruder(12171.40328)
  MoveL 1222 to (-5.96, -26.09, 60) mm, rotated rx -180 ry 0 rz 180 deg; joints [-163.733, -57.338, -93.242, 18.52, 61.866, -8.976]
  Call Extruder(12180.76837)
  MoveL 1223 to (0, -26.77, 60) mm, rotated rx -180 ry 0 rz 180 deg; joints [-164.103, -57.605, -92.307, 18.219, 61.174, -9.018]
  Call Extruder(12182.49841)
  MoveL 1224 to (1.1, -26.64, 60) mm, rotated rx 180 ry 0 rz 180 deg; joints [-164.132, -57.659, -92.122, 18.209, 61.044, -9.049]
  Call Extruder(12190.13349)
  MoveL 1225 to (5.96, -26.09, 60) mm, rotated rx 180 ry 0 rz 180 deg; joints [-164.258, -57.9, -91.299, 18.168, 60.472, -9.187]
  Call Extruder(12199.49829)
  MoveL 1226 to (11.61, -24.11, 60) mm, rotated rx 180 ry 0 rz 180 deg; joints [-164.201, -58.208, -90.271, 18.363, 59.797, -9.48]
  Call Extruder(12208.86320)
  MoveL 1227 to (16.69, -20.93, 60) mm, rotated rx 180 ry 0 rz 180 deg; joints [-163.944, -58.514, -89.272, 18.787, 59.184, -9.885]
  Call Extruder(12218.22841)
  MoveL 1228 to (20.93, -16.69, 60) mm, rotated rx 180 ry 0 rz 180 deg; joints [-163.508, -58.802, -88.352, 19.413, 58.663, -10.386]
  Call Extruder(12227.59333)
  MoveL 1229 to (24.12, -11.61, 60) mm, rotated rx 180 ry 0 rz 180 deg; joints [-162.92, -59.056, -87.555, 20.204, 58.261, -10.956]
  Call Extruder(12236.95812)
  MoveL 1230 to (26.09, -5.96, 60) mm, rotated rx -180 ry 0 rz -180 deg; joints [-162.209, -59.261, -86.918, 21.119, 57.996, -11.569]
  Call Extruder(12246.32322)
  MoveL 1231 to (26.77, 0, 60) mm, rotated rx -180 ry 0 rz -180 deg; joints [-161.41, -59.406, -86.472, 22.111, 57.881, -12.189]
  Call Extruder(12255.68833)
  MoveL 1232 to (26.09, 5.96, 60) mm, rotated rx -180 ry 0 rz 180 deg; joints [-160.556, -59.483, -86.239, 23.133, 57.921, -12.784]
  Call Extruder(12265.05313)
  MoveL 1233 to (24.12, 11.61, 60) mm, rotated rx 180 ry 0 rz 180 deg; joints [-159.683, -59.487, -86.227, 24.138, 58.111, -13.318]
  Call Extruder(12274.41804)
  MoveL 1234 to (20.93, 16.69, 60) mm, rotated rx -180 ry 0 rz 180 deg; joints [-158.826, -59.417, -86.44, 25.081, 58.441, -13.764]
  Call Extruder(12283.78325)
  MoveL 1235 to (16.69, 20.93, 60) mm, rotated rx -180 ry 0 rz 180 deg; joints [-158.019, -59.278, -86.865, 25.922, 58.894, -14.096]
  Call Extruder(12293.14816)
  MoveL 1236 to (11.61, 24.11, 60) mm, rotated rx -180 ry 0 rz 180 deg; joints [-157.299, -59.079, -87.484, 26.625, 59.447, -14.297]
  Call Extruder(12302.51297)
  MoveL 1237 to (5.96, 26.09, 60) mm, rotated rx 180 ry 0 rz -180 deg; joints [-156.697, -58.829, -88.267, 27.159, 60.071, -14.357]
  Call Extruder(12311.87807)
  MoveL 1238 to (0, 26.77, 60) mm, rotated rx 180 ry 0 rz 180 deg; joints [-156.245, -58.544, -89.176, 27.5, 60.738, -14.276]
  Call Extruder(12321.24317)
  MoveL 1239 to (-5.96, 26.09, 60) mm, rotated rx 180 ry 0 rz 180 deg; joints [-155.969, -58.239, -90.17, 27.63, 61.415, -14.06]
  Call Extruder(12330.60797)
  MoveL 1240 to (-11.61, 24.12, 60) mm, rotated rx 180 ry 0 rz 180 deg; joints [-155.891, -57.93, -91.197, 27.537, 62.072, -13.723]
  Call Extruder(12339.97289)
  MoveL 1241 to (-16.69, 20.93, 60) mm, rotated rx 180 ry 0 rz -180 deg; joints [-156.025, -57.633, -92.209, 27.218, 62.675, -13.284]
  Call Extruder(12349.33809)
  MoveL 1242 to (-20.93, 16.69, 60) mm, rotated rx 180 ry 0 rz 180 deg; joints [-156.374, -57.363, -93.154, 26.68, 63.198, -12.767]
